LIN {X 0,Y 100.527,Z 408.465,A -85,B 0,C 180,E1 -25391.818,E2 -25391.818} C_VEL
LIN {X 0,Y 102.586,Z 414.77,A -85,B 0,C 180,E1 -25385.896,E2 -25385.896} C_VEL
LIN {X 0,Y 105.943,Z 419.989,A -85,B 0,C 180,E1 -25379.998,E2 -25379.998} C_VEL
LIN {X 0,Y 110.426,Z 424.014,A -85,B 0,C 180,E1 -25374.52,E2 -25374.52} C_VEL
LIN {X 0,Y 116.041,Z 426.901,A -85,B 0,C 180,E1 -25369.53,E2 -25369.53} C_VEL
LIN {X 0,Y 120.304,Z 428.232,A -85,B 0,C 180,E1 -25366.485,E2 -25366.485} C_VEL
LIN {X 0,Y 124.925,Z 429.078,A -85,B 0,C 180,E1 -25363.661,E2 -25363.661} C_VEL
LIN {X 0,Y 131.477,Z 429.442,A -85,B 0,C 180,E1 -25360.34,E2 -25360.34} C_VEL
LIN {X 0,Y 140.786,Z 428.809,A -85,B 0,C 180,E1 -25356.461,E2 -25356.461} C_VEL
LIN {X 0,Y 148.981,Z 427.173,A -85,B 0,C 180,E1 -25353.679,E2 -25353.679} C_VEL
LIN {X 0,Y 158.987,Z 424.026,A -85,B 0,C 180,E1 -25350.904,E2 -25350.904} C_VEL
LIN {X 0,Y 169.115,Z 419.541,A -85,B 0,C 180,E1 -25348.564,E2 -25348.564} C_VEL
LIN {X 0,Y 167.944,Z 420.358,A -85,B 0,C 180,E1 -25347.788,E2 -25347.788} C_VEL
LIN {X 0,Y 157.475,Z 425.979,A -85,B 0,C 180,E1 -25345.656,E2 -25345.656} C_VEL
LIN {X 0,Y 148.742,Z 429.762,A -85,B 0,C 180,E1 -25343.443,E2 -25343.443} C_VEL
LIN {X 0,Y 139.769,Z 432.826,A -85,B 0,C 180,E1 -25340.691,E2 -25340.691} C_VEL
LIN {X 0,Y 134.979,Z 434.073,A -85,B 0,C 180,E1 -25339.334,E2 -25339.334} C_VEL
LIN {X 0,Y 126.203,Z 435.352,A -85,B 0,C 180,E1 -25337.386,E2 -25337.386} C_VEL
LIN {X 0,Y 117.725,Z 435.788,A -85,B 0,C 180,E1 -25335.033,E2 -25335.033} C_VEL
LIN {X 0,Y 113.512,Z 435.775,A -85,B 0,C 180,E1 -25333.009,E2 -25333.009} C_VEL
LIN {X 0,Y 105.631,Z 435.098,A -85,B 0,C 180,E1 -25326.787,E2 -25326.787} C_VEL
LIN {X 0,Y 99.678,Z 433.169,A -85,B 0,C 180,E1 -25319.577,E2 -25319.577} C_VEL
LIN {X 0,Y 96.026,Z 429.965,A -85,B 0,C 180,E1 -25311.469,E2 -25311.469} C_VEL
LIN {X 0,Y 94.866,Z 425.439,A -85,B 0,C 180,E1 -25302.844,E2 -25302.844} C_VEL
LIN {X 0,Y 95.674,Z 420.934,A -85,B 0,C 180,E1 -25296.329,E2 -25296.329} C_VEL
LIN {X 0,Y 96.226,Z 419.177,A -85,B 0,C 180,E1 -25294.191,E2 -25294.191} C_VEL
LIN {X 0,Y 95.972,Z 415.73,A -85,B 0,C 180,E1 -25291.052,E2 -25291.052} C_VEL
LIN {X 0,Y 95.262,Z 408.535,A -85,B 0,C 180,E1 -25285.772,E2 -25285.772} C_VEL
LIN {X 0,Y 95.129,Z 399.527,A -85,B 0,C 180,E1 -25280.435,E2 -25280.435} C_VEL
LIN {X 0,Y 95.647,Z 389.719,A -85,B 0,C 180,E1 -25275.746,E2 -25275.746} C_VEL
LIN {X 0,Y 96.578,Z 378.914,A -85,B 0,C 180,E1 -25271.723,E2 -25271.723} C_VEL
LIN {X 0,Y 97.631,Z 367.123,A -85,B 0,C 180,E1 -25268.354,E2 -25268.354} C_VEL
LIN {X 0,Y 98.64,Z 354.886,A -85,B 0,C 180,E1 -25265.819,E2 -25265.819} C_VEL
LIN {X 0,Y 99.244,Z 342.152,A -85,B 0,C 180,E1 -25264.016,E2 -25264.016} C_VEL
LIN {X 0,Y 100.899,Z 303.926,A -85,B 0,C 180,E1 -25259.798,E2 -25259.798} C_VEL
LIN {X 0,Y 99.621,Z 267.157,A -85,B 0,C 180,E1 -25255.645,E2 -25255.645} C_VEL
LIN {X 0,Y 99.558,Z 258.226,A -85,B 0,C 180,E1 -25254.646,E2 -25254.646} C_VEL
LIN {X 0,Y 97.627,Z 250.234,A -85,B 0,C 180,E1 -25253.451,E2 -25253.451} C_VEL
LIN {X 0,Y 95.667,Z 241.869,A -85,B 0,C 180,E1 -25247.279,E2 -25247.279} C_VEL
LIN {X 0,Y 93.662,Z 232.93,A -85,B 0,C 180,E1 -25239.981,E2 -25239.981} C_VEL
LIN {X 0,Y 93.575,Z 232.827,A -85,B 0,C 180,E1 -25231.72,E2 -25231.72} C_VEL
LIN {X 0,Y 93.665,Z 232.813,A -85,B 0,C 180,E1 -25225.797,E2 -25225.797} C_VEL
LIN {X 0,Y 93.69,Z 232.814,A -85,B 0,C 180,E1 -25222.031,E2 -25222.031} C_VEL
LIN {X 0,Y 94.087,Z 232.763,A -85,B 0,C 180,E1 -25212.951,E2 -25212.951} C_VEL
LIN {X 0,Y 94.195,Z 232.749,A -85,B 0,C 180,E1 -25208.584,E2 -25208.584} C_VEL
LIN {X 0,Y 94.786,Z 232.675,A -85,B 0,C 180,E1 -25200.002,E2 -25200.002} C_VEL
LIN {X 0,Y 94.17,Z 232.753,A -85,B 0,C 180,E1 -25191.418,E2 -25191.418} C_VEL
LIN {X 0,Y 94.018,Z 232.768,A -85,B 0,C 180,E1 -25186.339,E2 -25186.339} C_VEL
LIN {X 0,Y 93.685,Z 232.809,A -85,B 0,C 180,E1 -25177.973,E2 -25177.973} C_VEL
LIN {X 0,Y 93.617,Z 232.823,A -85,B 0,C 180,E1 -25173.231,E2 -25173.231} C_VEL
LIN {X 0,Y 93.607,Z 232.825,A -85,B 0,C 180,E1 -25165.672,E2 -25165.672} C_VEL
LIN {X 0,Y 93.625,Z 232.821,A -85,B 0,C 180,E1 -25157.503,E2 -25157.503} C_VEL
LIN {X 0,Y 93.623,Z 232.815,A -85,B 0,C 180,E1 -25151.355,E2 -25151.355} C_VEL
LIN {X 0,Y 93.609,Z 232.818,A -85,B 0,C 180,E1 -25144.328,E2 -25144.328} C_VEL
LIN {X 0,Y 93.665,Z 232.812,A -85,B 0,C 180,E1 -25135.794,E2 -25135.794} C_VEL
LIN {X 0,Y 93.689,Z 232.814,A -85,B 0,C 180,E1 -25132.025,E2 -25132.025} C_VEL
LIN {X 0,Y 94.088,Z 232.765,A -85,B 0,C 180,E1 -25122.946,E2 -25122.946} C_VEL
LIN {X 0,Y 94.197,Z 232.744,A -85,B 0,C 180,E1 -25118.579,E2 -25118.579} C_VEL
LIN {X 0,Y 94.794,Z 232.67,A -85,B 0,C 180,E1 -25109.997,E2 -25109.997} C_VEL
LIN {X 0,Y 94.209,Z 232.743,A -85,B 0,C 180,E1 -25101.416,E2 -25101.416} C_VEL
LIN {X 0,Y 94.045,Z 232.77,A -85,B 0,C 180,E1 -25096.276,E2 -25096.276} C_VEL
LIN {X 0,Y 93.692,Z 232.812,A -85,B 0,C 180,E1 -25087.969,E2 -25087.969} C_VEL
LIN {X 0,Y 93.813,Z 232.951,A -85,B 0,C 180,E1 -25080.549,E2 -25080.549} C_VEL
LIN {X 0,Y 94.861,Z 237.645,A -85,B 0,C 180,E1 -25076.331,E2 -25076.331} C_VEL
LIN {X 0,Y 95.705,Z 241.642,A -85,B 0,C 180,E1 -25073.185,E2 -25073.185} C_VEL
LIN {X 0,Y 100.113,Z 259.74,A -85,B 0,C 180,E1 -25070.488,E2 -25070.488} C_VEL
LIN {X 0,Y 101.197,Z 271.435,A -85,B 0,C 180,E1 -25069.044,E2 -25069.044} C_VEL
LIN {X 0,Y 97.514,Z 333.744,A -85,B 0,C 180,E1 -25061.785,E2 -25061.785} C_VEL
LIN {X 0,Y 96.446,Z 347.717,A -85,B 0,C 180,E1 -25059.273,E2 -25059.273} C_VEL
LIN {X 0,Y 95.268,Z 359.841,A -85,B 0,C 180,E1 -25056.166,E2 -25056.166} C_VEL
LIN {X 0,Y 94.062,Z 371.748,A -85,B 0,C 180,E1 -25052.089,E2 -25052.089} C_VEL
LIN {X 0,Y 93.221,Z 382.27,A -85,B 0,C 180,E1 -25047.499,E2 -25047.499} C_VEL
LIN {X 0,Y 92.756,Z 391.836,A -85,B 0,C 180,E1 -25042.26,E2 -25042.26} C_VEL
LIN {X 0,Y 92.8,Z 400.424,A -85,B 0,C 180,E1 -25036.497,E2 -25036.497} C_VEL
LIN {X 0,Y 93.861,Z 407.958,A -85,B 0,C 180,E1 -25030.304,E2 -25030.304} C_VEL
LIN {X 0,Y 96.102,Z 414.282,A -85,B 0,C 180,E1 -25024.192,E2 -25024.192} C_VEL
LIN {X 0,Y 99.787,Z 419.82,A -85,B 0,C 180,E1 -25017.98,E2 -25017.98} C_VEL
LIN {X 0,Y 104.629,Z 424.049,A -85,B 0,C 180,E1 -25012.278,E2 -25012.278} C_VEL
LIN {X 0,Y 108.524,Z 426.246,A -85,B 0,C 180,E1 -25008.796,E2 -25008.796} C_VEL
LIN {X 0,Y 112.895,Z 428.007,A -85,B 0,C 180,E1 -25005.579,E2 -25005.579} C_VEL
LIN {X 0,Y 117.979,Z 429.323,A -85,B 0,C 180,E1 -25002.392,E2 -25002.392} C_VEL
LIN {X 0,Y 126.464,Z 430.273,A -85,B 0,C 180,E1 -24998.15,E2 -24998.15} C_VEL
LIN {X 0,Y 133.801,Z 430.216,A -85,B 0,C 180,E1 -24995.151,E2 -24995.151} C_VEL
LIN {X 0,Y 143.305,Z 429.03,A -85,B 0,C 180,E1 -24991.98,E2 -24991.98} C_VEL
LIN {X 0,Y 152.344,Z 426.875,A -85,B 0,C 180,E1 -24989.504,E2 -24989.504} C_VEL
LIN {X 0,Y 156.663,Z 425.494,A -85,B 0,C 180,E1 -24988.471,E2 -24988.471} C_VEL
LIN {X 0,Y 144.639,Z 430.196,A -85,B 0,C 180,E1 -24985.696,E2 -24985.696} C_VEL
LIN {X 0,Y 133.24,Z 433.412,A -85,B 0,C 180,E1 -24982.301,E2 -24982.301} C_VEL
LIN {X 0,Y 122.723,Z 435.225,A -85,B 0,C 180,E1 -24978.117,E2 -24978.117} C_VEL
LIN {X 0,Y 113.512,Z 435.775,A -85,B 0,C 180,E1 -24973.009,E2 -24973.009} C_VEL
LIN {X 0,Y 109.506,Z 435.577,A -85,B 0,C 180,E1 -24970.776,E2 -24970.776} C_VEL
LIN {X 0,Y 102.13,Z 434.213,A -85,B 0,C 180,E1 -24967.256,E2 -24967.256} C_VEL
LIN {X 0,Y 95.497,Z 432.125,A -85,B 0,C 180,E1 -24963.169,E2 -24963.169} C_VEL
LIN {X 0,Y 92.799,Z 430.741,A -85,B 0,C 180,E1 -24960.084,E2 -24960.084} C_VEL
LIN {X 0,Y 89.119,Z 426.724,A -85,B 0,C 180,E1 -24950.789,E2 -24950.789} C_VEL
LIN {X 0,Y 88.499,Z 421.402,A -85,B 0,C 180,E1 -24941.454,E2 -24941.454} C_VEL
LIN {X 0,Y 89.676,Z 416.276,A -85,B 0,C 180,E1 -24934.498,E2 -24934.498} C_VEL
LIN {X 0,Y 89.047,Z 411.079,A -85,B 0,C 180,E1 -24930.003,E2 -24930.003} C_VEL
LIN {X 0,Y 88.409,Z 402.899,A -85,B 0,C 180,E1 -24924.301,E2 -24924.301} C_VEL
LIN {X 0,Y 88.508,Z 392.727,A -85,B 0,C 180,E1 -24918.553,E2 -24918.553} C_VEL
LIN {X 0,Y 89.198,Z 382.49,A -85,B 0,C 180,E1 -24913.996,E2 -24913.996} C_VEL
LIN {X 0,Y 90.216,Z 370.996,A -85,B 0,C 180,E1 -24910.003,E2 -24910.003} C_VEL
LIN {X 0,Y 91.441,Z 357.072,A -85,B 0,C 180,E1 -24906.507,E2 -24906.507} C_VEL
LIN {X 0,Y 92.057,Z 344.663,A -85,B 0,C 180,E1 -24904.421,E2 -24904.421} C_VEL
LIN {X 0,Y 93.823,Z 304.102,A -85,B 0,C 180,E1 -24899.536,E2 -24899.536} C_VEL
LIN {X 0,Y 92.573,Z 267.775,A -85,B 0,C 180,E1 -24895.12,E2 -24895.12} C_VEL
LIN {X 0,Y 92.653,Z 259.76,A -85,B 0,C 180,E1 -24894.166,E2 -24894.166} C_VEL
LIN {X 0,Y 90.29,Z 249.862,A -85,B 0,C 180,E1 -24892.583,E2 -24892.583} C_VEL
LIN {X 0,Y 88.272,Z 241.356,A -85,B 0,C 180,E1 -24885.774,E2 -24885.774} C_VEL
LIN {X 0,Y 86.553,Z 233.814,A -85,B 0,C 180,E1 -24878.989,E2 -24878.989} C_VEL
LIN {X 0,Y 86.53,Z 233.708,A -85,B 0,C 180,E1 -24874.651,E2 -24874.651} C_VEL
LIN {X 0,Y 86.579,Z 233.693,A -85,B 0,C 180,E1 -24866.767,E2 -24866.767} C_VEL
LIN {X 0,Y 86.643,Z 233.684,A -85,B 0,C 180,E1 -24858.935,E2 -24858.935} C_VEL
LIN {X 0,Y 86.965,Z 233.652,A -85,B 0,C 180,E1 -24854.033,E2 -24854.033} C_VEL
LIN {X 0,Y 87.103,Z 233.629,A -85,B 0,C 180,E1 -24849.289,E2 -24849.289} C_VEL
LIN {X 0,Y 87.713,Z 233.556,A -85,B 0,C 180,E1 -24840.002,E2 -24840.002} C_VEL
LIN {X 0,Y 87.08,Z 233.637,A -85,B 0,C 180,E1 -24830.713,E2 -24830.713} C_VEL
LIN {X 0,Y 86.925,Z 233.65,A -85,B 0,C 180,E1 -24825.965,E2 -24825.965} C_VEL
LIN {X 0,Y 86.638,Z 233.693,A -85,B 0,C 180,E1 -24821.069,E2 -24821.069} C_VEL
LIN {X 0,Y 86.579,Z 233.7,A -85,B 0,C 180,E1 -24813.233,E2 -24813.233} C_VEL
LIN {X 0,Y 86.531,Z 233.707,A -85,B 0,C 180,E1 -24804.305,E2 -24804.305} C_VEL
LIN {X 0,Y 86.553,Z 233.703,A -85,B 0,C 180,E1 -24796.947,E2 -24796.947} C_VEL
LIN {X 0,Y 86.548,Z 233.698,A -85,B 0,C 180,E1 -24790.509,E2 -24790.509} C_VEL
LIN {X 0,Y 86.556,Z 233.697,A -85,B 0,C 180,E1 -24784.632,E2 -24784.632} C_VEL
LIN {X 0,Y 86.581,Z 233.696,A -85,B 0,C 180,E1 -24776.765,E2 -24776.765} C_VEL
LIN {X 0,Y 86.658,Z 233.688,A -85,B 0,C 180,E1 -24768.926,E2 -24768.926} C_VEL
LIN {X 0,Y 86.966,Z 233.651,A -85,B 0,C 180,E1 -24764.027,E2 -24764.027} C_VEL
LIN {X 0,Y 87.105,Z 233.629,A -85,B 0,C 180,E1 -24759.283,E2 -24759.283} C_VEL
LIN {X 0,Y 87.721,Z 233.55,A -85,B 0,C 180,E1 -24749.997,E2 -24749.997} C_VEL
LIN {X 0,Y 87.115,Z 233.626,A -85,B 0,C 180,E1 -24740.712,E2 -24740.712} C_VEL
LIN {X 0,Y 86.949,Z 233.654,A -85,B 0,C 180,E1 -24735.909,E2 -24735.909} C_VEL
LIN {X 0,Y 86.662,Z 233.69,A -85,B 0,C 180,E1 -24731.068,E2 -24731.068} C_VEL
LIN {X 0,Y 86.708,Z 233.721,A -85,B 0,C 180,E1 -24721.757,E2 -24721.757} C_VEL
LIN {X 0,Y 86.974,Z 234.779,A -85,B 0,C 180,E1 -24720.331,E2 -24720.331} C_VEL
LIN {X 0,Y 88.541,Z 241.92,A -85,B 0,C 180,E1 -24714.05,E2 -24714.05} C_VEL
LIN {X 0,Y 93.165,Z 260.956,A -85,B 0,C 180,E1 -24710.987,E2 -24710.987} C_VEL
LIN {X 0,Y 94.057,Z 272.878,A -85,B 0,C 180,E1 -24709.439,E2 -24709.439} C_VEL
LIN {X 0,Y 90.386,Z 334.333,A -85,B 0,C 180,E1 -24701.646,E2 -24701.646} C_VEL
LIN {X 0,Y 89.315,Z 347.777,A -85,B 0,C 180,E1 -24699.011,E2 -24699.011} C_VEL
LIN {X 0,Y 88.063,Z 360.548,A -85,B 0,C 180,E1 -24695.448,E2 -24695.448} C_VEL
LIN {X 0,Y 86.936,Z 372.452,A -85,B 0,C 180,E1 -24691.019,E2 -24691.019} C_VEL
LIN {X 0,Y 86.193,Z 382.575,A -85,B 0,C 180,E1 -24686.238,E2 -24686.238} C_VEL
LIN {X 0,Y 85.855,Z 390.572,A -85,B 0,C 180,E1 -24681.612,E2 -24681.612} C_VEL
LIN {X 0,Y 86.125,Z 400.857,A -85,B 0,C 180,E1 -24674.168,E2 -24674.168} C_VEL
LIN {X 0,Y 87.827,Z 409.128,A -85,B 0,C 180,E1 -24666.892,E2 -24666.892} C_VEL
LIN {X 0,Y 90.949,Z 415.817,A -85,B 0,C 180,E1 -24659.998,E2 -24659.998} C_VEL
LIN {X 0,Y 95.39,Z 421.11,A -85,B 0,C 180,E1 -24653.653,E2 -24653.653} C_VEL
LIN {X 0,Y 101.091,Z 425.24,A -85,B 0,C 180,E1 -24647.96,E2 -24647.96} C_VEL
LIN {X 0,Y 105.481,Z 427.38,A -85,B 0,C 180,E1 -24644.541,E2 -24644.541} C_VEL
LIN {X 0,Y 111.809,Z 429.446,A -85,B 0,C 180,E1 -24640.543,E2 -24640.543} C_VEL
LIN {X 0,Y 121.658,Z 431.046,A -85,B 0,C 180,E1 -24635.765,E2 -24635.765} C_VEL
LIN {X 0,Y 126.882,Z 431.269,A -85,B 0,C 180,E1 -24633.695,E2 -24633.695} C_VEL
LIN {X 0,Y 137.831,Z 430.624,A -85,B 0,C 180,E1 -24630.095,E2 -24630.095} C_VEL
LIN {X 0,Y 142.117,Z 429.979,A -85,B 0,C 180,E1 -24628.902,E2 -24628.902} C_VEL
LIN {X 0,Y 140.774,Z 430.471,A -85,B 0,C 180,E1 -24628.074,E2 -24628.074} C_VEL
LIN {X 0,Y 129.039,Z 433.206,A -85,B 0,C 180,E1 -24624.785,E2 -24624.785} C_VEL
LIN {X 0,Y 118.12,Z 434.581,A -85,B 0,C 180,E1 -24620.671,E2 -24620.671} C_VEL
LIN {X 0,Y 108.003,Z 434.667,A -85,B 0,C 180,E1 -24615.247,E2 -24615.247} C_VEL
LIN {X 0,Y 100.128,Z 433.644,A -85,B 0,C 180,E1 -24609.179,E2 -24609.179} C_VEL
LIN {X 0,Y 93.747,Z 431.355,A -85,B 0,C 180,E1 -24601.656,E2 -24601.656} C_VEL
LIN {X 0,Y 92.799,Z 430.741,A -85,B 0,C 180,E1 -24600.084,E2 -24600.084} C_VEL
LIN {X 0,Y 90.51,Z 429.227,A -85,B 0,C 180,E1 -24596.832,E2 -24596.832} C_VEL
LIN {X 0,Y 86.053,Z 425.576,A -85,B 0,C 180,E1 -24591.595,E2 -24591.595} C_VEL
LIN {X 0,Y 82.643,Z 421.188,A -85,B 0,C 180,E1 -24585.977,E2 -24585.977} C_VEL
LIN {X 0,Y 82.108,Z 418.58,A -85,B 0,C 180,E1 -24582.287,E2 -24582.287} C_VEL
LIN {X 0,Y 83.036,Z 414.21,A -85,B 0,C 180,E1 -24576.076,E2 -24576.076} C_VEL
LIN {X 0,Y 83.145,Z 413.131,A -85,B 0,C 180,E1 -24574.852,E2 -24574.852} C_VEL
LIN {X 0,Y 82.097,Z 405.873,A -85,B 0,C 180,E1 -24568.777,E2 -24568.777} C_VEL
LIN {X 0,Y 81.633,Z 396.676,A -85,B 0,C 180,E1 -24562.584,E2 -24562.584} C_VEL
LIN {X 0,Y 81.996,Z 386.295,A -85,B 0,C 180,E1 -24557.001,E2 -24557.001} C_VEL
LIN {X 0,Y 82.86,Z 374.567,A -85,B 0,C 180,E1 -24552.097,E2 -24552.097} C_VEL
LIN {X 0,Y 83.967,Z 361.337,A -85,B 0,C 180,E1 -24548.031,E2 -24548.031} C_VEL
LIN {X 0,Y 84.765,Z 349.696,A -85,B 0,C 180,E1 -24545.512,E2 -24545.512} C_VEL
LIN {X 0,Y 86.102,Z 319.784,A -85,B 0,C 180,E1 -24541.349,E2 -24541.349} C_VEL
LIN {X 0,Y 86.708,Z 303.454,A -85,B 0,C 180,E1 -24539.23,E2 -24539.23} C_VEL
LIN {X 0,Y 85.561,Z 268.314,A -85,B 0,C 180,E1 -24534.582,E2 -24534.582} C_VEL
LIN {X 0,Y 85.542,Z 260.373,A -85,B 0,C 180,E1 -24533.547,E2 -24533.547} C_VEL
LIN {X 0,Y 82.924,Z 249.539,A -85,B 0,C 180,E1 -24531.665,E2 -24531.665} C_VEL
LIN {X 0,Y 80.902,Z 240.896,A -85,B 0,C 180,E1 -24524.028,E2 -24524.028} C_VEL
LIN {X 0,Y 79.486,Z 234.684,A -85,B 0,C 180,E1 -24517.876,E2 -24517.876} C_VEL
LIN {X 0,Y 79.477,Z 234.578,A -85,B 0,C 180,E1 -24507.845,E2 -24507.845} C_VEL
LIN {X 0,Y 79.51,Z 234.577,A -85,B 0,C 180,E1 -24500.708,E2 -24500.708} C_VEL
LIN {X 0,Y 79.837,Z 234.54,A -85,B 0,C 180,E1 -24494.477,E2 -24494.477} C_VEL
LIN {X 0,Y 79.989,Z 234.513,A -85,B 0,C 180,E1 -24490.123,E2 -24490.123} C_VEL
LIN {X 0,Y 80.64,Z 234.437,A -85,B 0,C 180,E1 -24480.002,E2 -24480.002} C_VEL
LIN {X 0,Y 79.962,Z 234.525,A -85,B 0,C 180,E1 -24469.878,E2 -24469.878} C_VEL
LIN {X 0,Y 79.738,Z 234.545,A -85,B 0,C 180,E1 -24464.67,E2 -24464.67} C_VEL
LIN {X 0,Y 79.506,Z 234.579,A -85,B 0,C 180,E1 -24459.296,E2 -24459.296} C_VEL
LIN {X 0,Y 79.478,Z 234.585,A -85,B 0,C 180,E1 -24452.153,E2 -24452.153} C_VEL
LIN {X 0,Y 79.441,Z 234.588,A -85,B 0,C 180,E1 -24442.763,E2 -24442.763} C_VEL
LIN {X 0,Y 79.461,Z 234.587,A -85,B 0,C 180,E1 -24434.966,E2 -24434.966} C_VEL
LIN {X 0,Y 79.447,Z 234.589,A -85,B 0,C 180,E1 -24427.24,E2 -24427.24} C_VEL
LIN {X 0,Y 79.48,Z 234.584,A -85,B 0,C 180,E1 -24417.846,E2 -24417.846} C_VEL
LIN {X 0,Y 79.518,Z 234.581,A -85,B 0,C 180,E1 -24410.699,E2 -24410.699} C_VEL
LIN {X 0,Y 79.838,Z 234.536,A -85,B 0,C 180,E1 -24404.472,E2 -24404.472} C_VEL
LIN {X 0,Y 79.99,Z 234.518,A -85,B 0,C 180,E1 -24400.117,E2 -24400.117} C_VEL
LIN {X 0,Y 80.649,Z 234.431,A -85,B 0,C 180,E1 -24389.996,E2 -24389.996} C_VEL
LIN {X 0,Y 79.998,Z 234.515,A -85,B 0,C 180,E1 -24379.877,E2 -24379.877} C_VEL
LIN {X 0,Y 79.764,Z 234.546,A -85,B 0,C 180,E1 -24374.669,E2 -24374.669} C_VEL
LIN {X 0,Y 79.527,Z 234.579,A -85,B 0,C 180,E1 -24369.296,E2 -24369.296} C_VEL
LIN {X 0,Y 79.677,Z 234.756,A -85,B 0,C 180,E1 -24362.426,E2 -24362.426} C_VEL
LIN {X 0,Y 81.142,Z 241.312,A -85,B 0,C 180,E1 -24355.733,E2 -24355.733} C_VEL
LIN {X 0,Y 81.37,Z 242.366,A -85,B 0,C 180,E1 -24354.903,E2 -24354.903} C_VEL
LIN {X 0,Y 86.246,Z 262.636,A -85,B 0,C 180,E1 -24351.415,E2 -24351.415} C_VEL
LIN {X 0,Y 87.016,Z 272.556,A -85,B 0,C 180,E1 -24350.008,E2 -24350.008} C_VEL
LIN {X 0,Y 83.263,Z 335.069,A -85,B 0,C 180,E1 -24341.377,E2 -24341.377} C_VEL
LIN {X 0,Y 82.113,Z 348.391,A -85,B 0,C 180,E1 -24338.523,E2 -24338.523} C_VEL
LIN {X 0,Y 81.013,Z 359.879,A -85,B 0,C 180,E1 -24335.078,E2 -24335.078} C_VEL
LIN {X 0,Y 79.964,Z 371.507,A -85,B 0,C 180,E1 -24330.519,E2 -24330.519} C_VEL
LIN {X 0,Y 79.257,Z 382.434,A -85,B 0,C 180,E1 -24324.907,E2 -24324.907} C_VEL
LIN {X 0,Y 78.947,Z 390.93,A -85,B 0,C 180,E1 -24319.499,E2 -24319.499} C_VEL
LIN {X 0,Y 79.536,Z 400.525,A -85,B 0,C 180,E1 -24312.087,E2 -24312.087} C_VEL
LIN {X 0,Y 81.361,Z 408.296,A -85,B 0,C 180,E1 -24304.953,E2 -24304.953} C_VEL
LIN {X 0,Y 85.331,Z 415.854,A -85,B 0,C 180,E1 -24296.872,E2 -24296.872} C_VEL
LIN {X 0,Y 89.703,Z 420.771,A -85,B 0,C 180,E1 -24290.983,E2 -24290.983} C_VEL
LIN {X 0,Y 95.944,Z 425.213,A -85,B 0,C 180,E1 -24285.057,E2 -24285.057} C_VEL
LIN {X 0,Y 103.095,Z 428.47,A -85,B 0,C 180,E1 -24280.069,E2 -24280.069} C_VEL
LIN {X 0,Y 108.366,Z 430.078,A -85,B 0,C 180,E1 -24277.098,E2 -24277.098} C_VEL
LIN {X 0,Y 118.859,Z 431.845,A -85,B 0,C 180,E1 -24272.494,E2 -24272.494} C_VEL
LIN {X 0,Y 128.984,Z 432.154,A -85,B 0,C 180,E1 -24269.065,E2 -24269.065} C_VEL
LIN {X 0,Y 128.114,Z 432.417,A -85,B 0,C 180,E1 -24268.305,E2 -24268.305} C_VEL
LIN {X 0,Y 119.296,Z 433.468,A -85,B 0,C 180,E1 -24265.569,E2 -24265.569} C_VEL
LIN {X 0,Y 108.537,Z 433.792,A -85,B 0,C 180,E1 -24260.992,E2 -24260.992} C_VEL
LIN {X 0,Y 99.039,Z 432.908,A -85,B 0,C 180,E1 -24255.207,E2 -24255.207} C_VEL
LIN {X 0,Y 91.16,Z 430.864,A -85,B 0,C 180,E1 -24248.084,E2 -24248.084} C_VEL
LIN {X 0,Y 85.449,Z 427.598,A -85,B 0,C 180,E1 -24239.573,E2 -24239.573} C_VEL
LIN {X 0,Y 82.404,Z 423.04,A -85,B 0,C 180,E1 -24229.95,E2 -24229.95} C_VEL
LIN {X 0,Y 82.108,Z 418.58,A -85,B 0,C 180,E1 -24222.287,E2 -24222.287} C_VEL
LIN {X 0,Y 81.96,Z 416.788,A -85,B 0,C 180,E1 -24219.899,E2 -24219.899} C_VEL
LIN {X 0,Y 81.28,Z 414.6,A -85,B 0,C 180,E1 -24217.675,E2 -24217.675} C_VEL
LIN {X 0,Y 79.644,Z 410.864,A -85,B 0,C 180,E1 -24214.59,E2 -24214.59} C_VEL
LIN {X 0,Y 75.525,Z 400.581,A -85,B 0,C 180,E1 -24207.668,E2 -24207.668} C_VEL
LIN {X 0,Y 75.066,Z 397.473,A -85,B 0,C 180,E1 -24205.585,E2 -24205.585} C_VEL
LIN {X 0,Y 75.076,Z 387.142,A -85,B 0,C 180,E1 -24199.213,E2 -24199.213} C_VEL
LIN {X 0,Y 75.735,Z 375.961,A -85,B 0,C 180,E1 -24193.84,E2 -24193.84} C_VEL
LIN {X 0,Y 76.669,Z 364.055,A -85,B 0,C 180,E1 -24189.549,E2 -24189.549} C_VEL
LIN {X 0,Y 77.501,Z 352.51,A -85,B 0,C 180,E1 -24186.516,E2 -24186.516} C_VEL
LIN {X 0,Y 78.112,Z 339.079,A -85,B 0,C 180,E1 -24184.129,E2 -24184.129} C_VEL
LIN {X 0,Y 79.659,Z 304.435,A -85,B 0,C 180,E1 -24179.153,E2 -24179.153} C_VEL
LIN {X 0,Y 78.522,Z 268.388,A -85,B 0,C 180,E1 -24173.937,E2 -24173.937} C_VEL
LIN {X 0,Y 78.489,Z 261.196,A -85,B 0,C 180,E1 -24172.893,E2 -24172.893} C_VEL
LIN {X 0,Y 75.592,Z 249.161,A -85,B 0,C 180,E1 -24170.609,E2 -24170.609} C_VEL
LIN {X 0,Y 73.516,Z 240.36,A -85,B 0,C 180,E1 -24162.008,E2 -24162.008} C_VEL
LIN {X 0,Y 72.385,Z 235.556,A -85,B 0,C 180,E1 -24156.624,E2 -24156.624} C_VEL
LIN {X 0,Y 72.372,Z 235.467,A -85,B 0,C 180,E1 -24149.051,E2 -24149.051} C_VEL
LIN {X 0,Y 72.39,Z 235.468,A -85,B 0,C 180,E1 -24142.854,E2 -24142.854} C_VEL
LIN {X 0,Y 72.732,Z 235.425,A -85,B 0,C 180,E1 -24134.937,E2 -24134.937} C_VEL
LIN {X 0,Y 72.875,Z 235.399,A -85,B 0,C 180,E1 -24131.123,E2 -24131.123} C_VEL
LIN {X 0,Y 73.566,Z 235.318,A -85,B 0,C 180,E1 -24120.003,E2 -24120.003} C_VEL
LIN {X 0,Y 72.853,Z 235.41,A -85,B 0,C 180,E1 -24108.879,E2 -24108.879} C_VEL
LIN {X 0,Y 72.567,Z 235.443,A -85,B 0,C 180,E1 -24103.112,E2 -24103.112} C_VEL
LIN {X 0,Y 72.387,Z 235.459,A -85,B 0,C 180,E1 -24097.151,E2 -24097.151} C_VEL
LIN {X 0,Y 72.37,Z 235.468,A -85,B 0,C 180,E1 -24090.918,E2 -24090.918} C_VEL
LIN {X 0,Y 72.329,Z 235.476,A -85,B 0,C 180,E1 -24084.341,E2 -24084.341} C_VEL
LIN {X 0,Y 72.304,Z 235.477,A -85,B 0,C 180,E1 -24077.129,E2 -24077.129} C_VEL
LIN {X 0,Y 72.354,Z 235.471,A -85,B 0,C 180,E1 -24069.011,E2 -24069.011} C_VEL
LIN {X 0,Y 72.333,Z 235.473,A -85,B 0,C 180,E1 -24065.654,E2 -24065.654} C_VEL
LIN {X 0,Y 72.387,Z 235.468,A -85,B 0,C 180,E1 -24059.037,E2 -24059.037} C_VEL
LIN {X 0,Y 72.395,Z 235.463,A -85,B 0,C 180,E1 -24052.845,E2 -24052.845} C_VEL
LIN {X 0,Y 72.753,Z 235.417,A -85,B 0,C 180,E1 -24044.993,E2 -24044.993} C_VEL
LIN {X 0,Y 72.876,Z 235.406,A -85,B 0,C 180,E1 -24041.116,E2 -24041.116} C_VEL
LIN {X 0,Y 73.575,Z 235.312,A -85,B 0,C 180,E1 -24029.996,E2 -24029.996} C_VEL
LIN {X 0,Y 72.883,Z 235.404,A -85,B 0,C 180,E1 -24018.877,E2 -24018.877} C_VEL
LIN {X 0,Y 72.586,Z 235.437,A -85,B 0,C 180,E1 -24013.11,E2 -24013.11} C_VEL
LIN {X 0,Y 72.567,Z 235.569,A -85,B 0,C 180,E1 -24003.773,E2 -24003.773} C_VEL
LIN {X 0,Y 73.029,Z 237.535,A -85,B 0,C 180,E1 -24001.234,E2 -24001.234} C_VEL
LIN {X 0,Y 74.194,Z 242.699,A -85,B 0,C 180,E1 -23995.933,E2 -23995.933} C_VEL
LIN {X 0,Y 79.335,Z 264.278,A -85,B 0,C 180,E1 -23991.874,E2 -23991.874} C_VEL
LIN {X 0,Y 79.893,Z 273.059,A -85,B 0,C 180,E1 -23990.524,E2 -23990.524} C_VEL
LIN {X 0,Y 76.195,Z 334.708,A -85,B 0,C 180,E1 -23981.263,E2 -23981.263} C_VEL
LIN {X 0,Y 75.091,Z 347.518,A -85,B 0,C 180,E1 -23978.317,E2 -23978.317} C_VEL
LIN {X 0,Y 73.926,Z 359.791,A -85,B 0,C 180,E1 -23974.321,E2 -23974.321} C_VEL
LIN {X 0,Y 72.883,Z 372.355,A -85,B 0,C 180,E1 -23968.822,E2 -23968.822} C_VEL
LIN {X 0,Y 72.315,Z 384.067,A -85,B 0,C 180,E1 -23962.12,E2 -23962.12} C_VEL
LIN {X 0,Y 72.451,Z 395.051,A -85,B 0,C 180,E1 -23954.047,E2 -23954.047} C_VEL
LIN {X 0,Y 74.106,Z 404.498,A -85,B 0,C 180,E1 -23945.439,E2 -23945.439} C_VEL
LIN {X 0,Y 77.82,Z 412.82,A -85,B 0,C 180,E1 -23936.764,E2 -23936.764} C_VEL
LIN {X 0,Y 82.314,Z 418.513,A -85,B 0,C 180,E1 -23930.166,E2 -23930.166} C_VEL
LIN {X 0,Y 89.104,Z 423.897,A -85,B 0,C 180,E1 -23923.399,E2 -23923.399} C_VEL
LIN {X 0,Y 95.903,Z 427.478,A -85,B 0,C 180,E1 -23918.503,E2 -23918.503} C_VEL
LIN {X 0,Y 101.339,Z 429.524,A -85,B 0,C 180,E1 -23915.409,E2 -23915.409} C_VEL
LIN {X 0,Y 107.145,Z 431.077,A -85,B 0,C 180,E1 -23912.665,E2 -23912.665} C_VEL
LIN {X 0,Y 113.45,Z 432.245,A -85,B 0,C 180,E1 -23910.147,E2 -23910.147} C_VEL
LIN {X 0,Y 115.46,Z 432.721,A -85,B 0,C 180,E1 -23908.453,E2 -23908.453} C_VEL
LIN {X 0,Y 104.276,Z 432.624,A -85,B 0,C 180,E1 -23903.98,E2 -23903.98} C_VEL
LIN {X 0,Y 94.273,Z 431.367,A -85,B 0,C 180,E1 -23898.206,E2 -23898.206} C_VEL
LIN {X 0,Y 85.882,Z 428.907,A -85,B 0,C 180,E1 -23890.898,E2 -23890.898} C_VEL
LIN {X 0,Y 79.65,Z 425.291,A -85,B 0,C 180,E1 -23881.97,E2 -23881.97} C_VEL
LIN {X 0,Y 76.23,Z 420.334,A -85,B 0,C 180,E1 -23871.644,E2 -23871.644} C_VEL
LIN {X 0,Y 75.807,Z 415.511,A -85,B 0,C 180,E1 -23863.089,E2 -23863.089} C_VEL
LIN {X 0,Y 76.716,Z 410.967,A -85,B 0,C 180,E1 -23856.579,E2 -23856.579} C_VEL
LIN {X 0,Y 75.774,Z 405.137,A -85,B 0,C 180,E1 -23851.332,E2 -23851.332} C_VEL
LIN {X 0,Y 75.066,Z 397.473,A -85,B 0,C 180,E1 -23845.585,E2 -23845.585} C_VEL
LIN {X 0,Y 74.33,Z 392.909,A -85,B 0,C 180,E1 -23842.82,E2 -23842.82} C_VEL
LIN {X 0,Y 72.905,Z 388.046,A -85,B 0,C 180,E1 -23840.423,E2 -23840.423} C_VEL
LIN {X 0,Y 69.477,Z 376.059,A -85,B 0,C 180,E1 -23835.365,E2 -23835.365} C_VEL
LIN {X 0,Y 69.165,Z 370.632,A -85,B 0,C 180,E1 -23833.148,E2 -23833.148} C_VEL
LIN {X 0,Y 70.01,Z 359.201,A -85,B 0,C 180,E1 -23829.05,E2 -23829.05} C_VEL
LIN {X 0,Y 70.722,Z 347.421,A -85,B 0,C 180,E1 -23826.028,E2 -23826.028} C_VEL
LIN {X 0,Y 72.581,Z 304.67,A -85,B 0,C 180,E1 -23818.971,E2 -23818.971} C_VEL
LIN {X 0,Y 71.485,Z 268.942,A -85,B 0,C 180,E1 -23813.324,E2 -23813.324} C_VEL
LIN {X 0,Y 71.477,Z 262.238,A -85,B 0,C 180,E1 -23812.269,E2 -23812.269} C_VEL
LIN {X 0,Y 68.247,Z 248.92,A -85,B 0,C 180,E1 -23809.475,E2 -23809.475} C_VEL
LIN {X 0,Y 66.128,Z 239.886,A -85,B 0,C 180,E1 -23799.622,E2 -23799.622} C_VEL
LIN {X 0,Y 65.267,Z 236.437,A -85,B 0,C 180,E1 -23795.132,E2 -23795.132} C_VEL
LIN {X 0,Y 65.257,Z 236.357,A -85,B 0,C 180,E1 -23790.516,E2 -23790.516} C_VEL
LIN {X 0,Y 65.234,Z 236.354,A -85,B 0,C 180,E1 -23785.53,E2 -23785.53} C_VEL
LIN {X 0,Y 65.632,Z 236.309,A -85,B 0,C 180,E1 -23775.496,E2 -23775.496} C_VEL
LIN {X 0,Y 65.768,Z 236.288,A -85,B 0,C 180,E1 -23772.343,E2 -23772.343} C_VEL
LIN {X 0,Y 66.489,Z 236.199,A -85,B 0,C 180,E1 -23760.003,E2 -23760.003} C_VEL
LIN {X 0,Y 65.749,Z 236.292,A -85,B 0,C 180,E1 -23747.659,E2 -23747.659} C_VEL
LIN {X 0,Y 65.374,Z 236.342,A -85,B 0,C 180,E1 -23741.188,E2 -23741.188} C_VEL
LIN {X 0,Y 65.24,Z 236.356,A -85,B 0,C 180,E1 -23734.479,E2 -23734.479} C_VEL
LIN {X 0,Y 65.208,Z 236.355,A -85,B 0,C 180,E1 -23727.395,E2 -23727.395} C_VEL
LIN {X 0,Y 65.238,Z 236.352,A -85,B 0,C 180,E1 -23718.939,E2 -23718.939} C_VEL
LIN {X 0,Y 65.262,Z 236.349,A -85,B 0,C 180,E1 -23710.245,E2 -23710.245} C_VEL
LIN {X 0,Y 65.255,Z 236.355,A -85,B 0,C 180,E1 -23700.509,E2 -23700.509} C_VEL
LIN {X 0,Y 65.244,Z 236.35,A -85,B 0,C 180,E1 -23695.518,E2 -23695.518} C_VEL
LIN {X 0,Y 65.647,Z 236.3,A -85,B 0,C 180,E1 -23685.536,E2 -23685.536} C_VEL
LIN {X 0,Y 65.777,Z 236.292,A -85,B 0,C 180,E1 -23682.334,E2 -23682.334} C_VEL
LIN {X 0,Y 66.499,Z 236.193,A -85,B 0,C 180,E1 -23669.996,E2 -23669.996} C_VEL
LIN {X 0,Y 65.782,Z 236.291,A -85,B 0,C 180,E1 -23657.658,E2 -23657.658} C_VEL
LIN {X 0,Y 65.4,Z 236.337,A -85,B 0,C 180,E1 -23651.188,E2 -23651.188} C_VEL
LIN {X 0,Y 65.421,Z 236.379,A -85,B 0,C 180,E1 -23645.396,E2 -23645.396} C_VEL
LIN {X 0,Y 65.822,Z 237.852,A -85,B 0,C 180,E1 -23643.009,E2 -23643.009} C_VEL
LIN {X 0,Y 67.04,Z 243.06,A -85,B 0,C 180,E1 -23637.051,E2 -23637.051} C_VEL
LIN {X 0,Y 72.333,Z 265.182,A -85,B 0,C 180,E1 -23632.473,E2 -23632.473} C_VEL
LIN {X 0,Y 72.854,Z 273.008,A -85,B 0,C 180,E1 -23631.17,E2 -23631.17} C_VEL
LIN {X 0,Y 69.08,Z 334.498,A -85,B 0,C 180,E1 -23620.911,E2 -23620.911} C_VEL
LIN {X 0,Y 68.037,Z 347.057,A -85,B 0,C 180,E1 -23617.78,E2 -23617.78} C_VEL
LIN {X 0,Y 66.87,Z 360.105,A -85,B 0,C 180,E1 -23613.143,E2 -23613.143} C_VEL
LIN {X 0,Y 65.881,Z 372.862,A -85,B 0,C 180,E1 -23606.951,E2 -23606.951} C_VEL
LIN {X 0,Y 65.514,Z 383.264,A -85,B 0,C 180,E1 -23600.401,E2 -23600.401} C_VEL
LIN {X 0,Y 65.872,Z 393.444,A -85,B 0,C 180,E1 -23592.318,E2 -23592.318} C_VEL
LIN {X 0,Y 67.82,Z 403.279,A -85,B 0,C 180,E1 -23582.967,E2 -23582.967} C_VEL
LIN {X 0,Y 71.602,Z 411.295,A -85,B 0,C 180,E1 -23574.364,E2 -23574.364} C_VEL
LIN {X 0,Y 76.964,Z 417.817,A -85,B 0,C 180,E1 -23566.801,E2 -23566.801} C_VEL
LIN {X 0,Y 83.714,Z 423.178,A -85,B 0,C 180,E1 -23560.376,E2 -23560.376} C_VEL
LIN {X 0,Y 91.594,Z 427.378,A -85,B 0,C 180,E1 -23555.033,E2 -23555.033} C_VEL
LIN {X 0,Y 102.609,Z 431.141,A -85,B 0,C 180,E1 -23549.697,E2 -23549.697} C_VEL
LIN {X 0,Y 103.671,Z 431.422,A -85,B 0,C 180,E1 -23549.275,E2 -23549.275} C_VEL
LIN {X 0,Y 102.028,Z 431.437,A -85,B 0,C 180,E1 -23547.937,E2 -23547.937} C_VEL
LIN {X 0,Y 94.901,Z 430.59,A -85,B 0,C 180,E1 -23544.554,E2 -23544.554} C_VEL
LIN {X 0,Y 85.095,Z 428.367,A -85,B 0,C 180,E1 -23538.018,E2 -23538.018} C_VEL
LIN {X 0,Y 77.175,Z 424.947,A -85,B 0,C 180,E1 -23529.607,E2 -23529.607} C_VEL
LIN {X 0,Y 71.76,Z 420.346,A -85,B 0,C 180,E1 -23519.324,E2 -23519.324} C_VEL
LIN {X 0,Y 69.595,Z 414.279,A -85,B 0,C 180,E1 -23507.639,E2 -23507.639} C_VEL
LIN {X 0,Y 70.293,Z 408.727,A -85,B 0,C 180,E1 -23498.629,E2 -23498.629} C_VEL
LIN {X 0,Y 69.942,Z 405.996,A -85,B 0,C 180,E1 -23495.771,E2 -23495.771} C_VEL
LIN {X 0,Y 68.691,Z 397.36,A -85,B 0,C 180,E1 -23488.538,E2 -23488.538} C_VEL
LIN {X 0,Y 68.358,Z 386.481,A -85,B 0,C 180,E1 -23481.133,E2 -23481.133} C_VEL
LIN {X 0,Y 68.866,Z 375.36,A -85,B 0,C 180,E1 -23475.223,E2 -23475.223} C_VEL
LIN {X 0,Y 69.165,Z 370.632,A -85,B 0,C 180,E1 -23473.148,E2 -23473.148} C_VEL
LIN {X 0,Y 68.836,Z 365.233,A -85,B 0,C 180,E1 -23471.165,E2 -23471.165} C_VEL
LIN {X 0,Y 67.581,Z 359.728,A -85,B 0,C 180,E1 -23469.557,E2 -23469.557} C_VEL
LIN {X 0,Y 64.193,Z 346.594,A -85,B 0,C 180,E1 -23466.538,E2 -23466.538} C_VEL
LIN {X 0,Y 63.877,Z 340.779,A -85,B 0,C 180,E1 -23465.378,E2 -23465.378} C_VEL
LIN {X 0,Y 65.474,Z 304.169,A -85,B 0,C 180,E1 -23458.808,E2 -23458.808} C_VEL
LIN {X 0,Y 64.468,Z 268.165,A -85,B 0,C 180,E1 -23452.421,E2 -23452.421} C_VEL
LIN {X 0,Y 64.4,Z 262.953,A -85,B 0,C 180,E1 -23451.485,E2 -23451.485} C_VEL
LIN {X 0,Y 60.871,Z 248.611,A -85,B 0,C 180,E1 -23448.147,E2 -23448.147} C_VEL
LIN {X 0,Y 59.414,Z 242.323,A -85,B 0,C 180,E1 -23440.59,E2 -23440.59} C_VEL
LIN {X 0,Y 58.182,Z 237.334,A -85,B 0,C 180,E1 -23433.669,E2 -23433.669} C_VEL
LIN {X 0,Y 58.15,Z 237.237,A -85,B 0,C 180,E1 -23428.914,E2 -23428.914} C_VEL
LIN {X 0,Y 58.522,Z 237.194,A -85,B 0,C 180,E1 -23416.128,E2 -23416.128} C_VEL
LIN {X 0,Y 58.813,Z 237.159,A -85,B 0,C 180,E1 -23406.866,E2 -23406.866} C_VEL
LIN {X 0,Y 59.379,Z 237.084,A -85,B 0,C 180,E1 -23400.003,E2 -23400.003} C_VEL
LIN {X 0,Y 58.793,Z 237.153,A -85,B 0,C 180,E1 -23393.138,E2 -23393.138} C_VEL
LIN {X 0,Y 58.511,Z 237.19,A -85,B 0,C 180,E1 -23383.909,E2 -23383.909} C_VEL
LIN {X 0,Y 58.151,Z 237.239,A -85,B 0,C 180,E1 -23371.094,E2 -23371.094} C_VEL
LIN {X 0,Y 58.065,Z 237.25,A -85,B 0,C 180,E1 -23362.762,E2 -23362.762} C_VEL
LIN {X 0,Y 58.087,Z 237.244,A -85,B 0,C 180,E1 -23353.457,E2 -23353.457} C_VEL
LIN {X 0,Y 58.069,Z 237.252,A -85,B 0,C 180,E1 -23347.232,E2 -23347.232} C_VEL
LIN {X 0,Y 58.153,Z 237.242,A -85,B 0,C 180,E1 -23338.903,E2 -23338.903} C_VEL
LIN {X 0,Y 58.533,Z 237.185,A -85,B 0,C 180,E1 -23326.16,E2 -23326.16} C_VEL
LIN {X 0,Y 58.816,Z 237.151,A -85,B 0,C 180,E1 -23316.858,E2 -23316.858} C_VEL
LIN {X 0,Y 59.391,Z 237.078,A -85,B 0,C 180,E1 -23309.995,E2 -23309.995} C_VEL
LIN {X 0,Y 58.822,Z 237.153,A -85,B 0,C 180,E1 -23303.133,E2 -23303.133} C_VEL
LIN {X 0,Y 58.532,Z 237.187,A -85,B 0,C 180,E1 -23293.845,E2 -23293.845} C_VEL
LIN {X 0,Y 58.34,Z 237.277,A -85,B 0,C 180,E1 -23286.946,E2 -23286.946} C_VEL
LIN {X 0,Y 58.885,Z 239.417,A -85,B 0,C 180,E1 -23283.407,E2 -23283.407} C_VEL
LIN {X 0,Y 59.873,Z 243.508,A -85,B 0,C 180,E1 -23278.357,E2 -23278.357} C_VEL
LIN {X 0,Y 65.268,Z 265.646,A -85,B 0,C 180,E1 -23273.199,E2 -23273.199} C_VEL
LIN {X 0,Y 65.782,Z 273.424,A -85,B 0,C 180,E1 -23271.744,E2 -23271.744} C_VEL
LIN {X 0,Y 61.992,Z 334.488,A -85,B 0,C 180,E1 -23260.41,E2 -23260.41} C_VEL
LIN {X 0,Y 60.968,Z 346.859,A -85,B 0,C 180,E1 -23257.029,E2 -23257.029} C_VEL
LIN {X 0,Y 59.921,Z 359.052,A -85,B 0,C 180,E1 -23252.308,E2 -23252.308} C_VEL
LIN {X 0,Y 59.053,Z 371.676,A -85,B 0,C 180,E1 -23245.554,E2 -23245.554} C_VEL
LIN {X 0,Y 58.881,Z 382.659,A -85,B 0,C 180,E1 -23237.943,E2 -23237.943} C_VEL
LIN {X 0,Y 59.623,Z 393.561,A -85,B 0,C 180,E1 -23228.47,E2 -23228.47} C_VEL
LIN {X 0,Y 61.723,Z 401.899,A -85,B 0,C 180,E1 -23219.997,E2 -23219.997} C_VEL
LIN {X 0,Y 66.034,Z 410.187,A -85,B 0,C 180,E1 -23210.811,E2 -23210.811} C_VEL
LIN {X 0,Y 71.93,Z 417.049,A -85,B 0,C 180,E1 -23202.953,E2 -23202.953} C_VEL
LIN {X 0,Y 79.251,Z 422.633,A -85,B 0,C 180,E1 -23196.478,E2 -23196.478} C_VEL
LIN {X 0,Y 88.627,Z 427.561,A -85,B 0,C 180,E1 -23190.73,E2 -23190.73} C_VEL
LIN {X 0,Y 91.735,Z 428.825,A -85,B 0,C 180,E1 -23189.223,E2 -23189.223} C_VEL
LIN {X 0,Y 91.076,Z 428.887,A -85,B 0,C 180,E1 -23188.089,E2 -23188.089} C_VEL
LIN {X 0,Y 80.711,Z 426.255,A -85,B 0,C 180,E1 -23181.604,E2 -23181.604} C_VEL
LIN {X 0,Y 72.15,Z 422.492,A -85,B 0,C 180,E1 -23172.994,E2 -23172.994} C_VEL
LIN {X 0,Y 66.017,Z 417.244,A -85,B 0,C 180,E1 -23161.602,E2 -23161.602} C_VEL
LIN {X 0,Y 63.598,Z 411.064,A -85,B 0,C 180,E1 -23149.366,E2 -23149.366} C_VEL
LIN {X 0,Y 64.115,Z 405.014,A -85,B 0,C 180,E1 -23139.393,E2 -23139.393} C_VEL
LIN {X 0,Y 62.452,Z 396.602,A -85,B 0,C 180,E1 -23131.617,E2 -23131.617} C_VEL
LIN {X 0,Y 61.702,Z 386.984,A -85,B 0,C 180,E1 -23124.285,E2 -23124.285} C_VEL
LIN {X 0,Y 61.883,Z 377.798,A -85,B 0,C 180,E1 -23118.541,E2 -23118.541} C_VEL
LIN {X 0,Y 62.52,Z 366.017,A -85,B 0,C 180,E1 -23112.842,E2 -23112.842} C_VEL
LIN {X 0,Y 63.403,Z 353.703,A -85,B 0,C 180,E1 -23108.463,E2 -23108.463} C_VEL
LIN {X 0,Y 63.877,Z 340.779,A -85,B 0,C 180,E1 -23105.378,E2 -23105.378} C_VEL
LIN {X 0,Y 63.57,Z 335.008,A -85,B 0,C 180,E1 -23104.327,E2 -23104.327} C_VEL
LIN {X 0,Y 58.654,Z 316.091,A -85,B 0,C 180,E1 -23101.043,E2 -23101.043} C_VEL
LIN {X 0,Y 58.208,Z 310.293,A -85,B 0,C 180,E1 -23099.918,E2 -23099.918} C_VEL
LIN {X 0,Y 58.281,Z 302.57,A -85,B 0,C 180,E1 -23098.396,E2 -23098.396} C_VEL
LIN {X 0,Y 57.468,Z 267.619,A -85,B 0,C 180,E1 -23091.451,E2 -23091.451} C_VEL
LIN {X 0,Y 57.33,Z 263.567,A -85,B 0,C 180,E1 -23090.629,E2 -23090.629} C_VEL
LIN {X 0,Y 53.545,Z 248.405,A -85,B 0,C 180,E1 -23086.627,E2 -23086.627} C_VEL
LIN {X 0,Y 52.022,Z 241.899,A -85,B 0,C 180,E1 -23077.673,E2 -23077.673} C_VEL
LIN {X 0,Y 51.13,Z 238.216,A -85,B 0,C 180,E1 -23071.608,E2 -23071.608} C_VEL
LIN {X 0,Y 51.389,Z 238.079,A -85,B 0,C 180,E1 -23056.822,E2 -23056.822} C_VEL
LIN {X 0,Y 51.688,Z 238.044,A -85,B 0,C 180,E1 -23047.818,E2 -23047.818} C_VEL
LIN {X 0,Y 52.262,Z 237.97,A -85,B 0,C 180,E1 -23040.004,E2 -23040.004} C_VEL
LIN {X 0,Y 51.67,Z 238.042,A -85,B 0,C 180,E1 -23032.186,E2 -23032.186} C_VEL
LIN {X 0,Y 51.381,Z 238.08,A -85,B 0,C 180,E1 -23023.211,E2 -23023.211} C_VEL
LIN {X 0,Y 51.021,Z 238.122,A -85,B 0,C 180,E1 -23015.595,E2 -23015.595} C_VEL
LIN {X 0,Y 51.044,Z 238.124,A -85,B 0,C 180,E1 -23005.691,E2 -23005.691} C_VEL
LIN {X 0,Y 51.05,Z 238.126,A -85,B 0,C 180,E1 -22996.506,E2 -22996.506} C_VEL
LIN {X 0,Y 51.051,Z 238.12,A -85,B 0,C 180,E1 -22993.489,E2 -22993.489} C_VEL
LIN {X 0,Y 51.069,Z 238.114,A -85,B 0,C 180,E1 -22983.392,E2 -22983.392} C_VEL
LIN {X 0,Y 51.025,Z 238.12,A -85,B 0,C 180,E1 -22974.4,E2 -22974.4} C_VEL
LIN {X 0,Y 51.478,Z 238.064,A -85,B 0,C 180,E1 -22965.84,E2 -22965.84} C_VEL
LIN {X 0,Y 51.692,Z 238.037,A -85,B 0,C 180,E1 -22957.808,E2 -22957.808} C_VEL
LIN {X 0,Y 52.276,Z 237.964,A -85,B 0,C 180,E1 -22949.995,E2 -22949.995} C_VEL
LIN {X 0,Y 51.698,Z 238.037,A -85,B 0,C 180,E1 -22942.181,E2 -22942.181} C_VEL
LIN {X 0,Y 51.433,Z 238.071,A -85,B 0,C 180,E1 -22933.025,E2 -22933.025} C_VEL
LIN {X 0,Y 51.306,Z 238.176,A -85,B 0,C 180,E1 -22928.88,E2 -22928.88} C_VEL
LIN {X 0,Y 51.643,Z 239.659,A -85,B 0,C 180,E1 -22925.899,E2 -22925.899} C_VEL
LIN {X 0,Y 52.64,Z 243.799,A -85,B 0,C 180,E1 -22919.95,E2 -22919.95} C_VEL
LIN {X 0,Y 56.67,Z 259.976,A -85,B 0,C 180,E1 -22915.505,E2 -22915.505} C_VEL
LIN {X 0,Y 58.396,Z 268.11,A -85,B 0,C 180,E1 -22913.608,E2 -22913.608} C_VEL
LIN {X 0,Y 58.71,Z 273.656,A -85,B 0,C 180,E1 -22912.467,E2 -22912.467} C_VEL
LIN {X 0,Y 54.948,Z 333.835,A -85,B 0,C 180,E1 -22899.871,E2 -22899.871} C_VEL
LIN {X 0,Y 53.92,Z 346.601,A -85,B 0,C 180,E1 -22895.963,E2 -22895.963} C_VEL
LIN {X 0,Y 52.859,Z 360.105,A -85,B 0,C 180,E1 -22889.902,E2 -22889.902} C_VEL
LIN {X 0,Y 52.276,Z 371.836,A -85,B 0,C 180,E1 -22882.719,E2 -22882.719} C_VEL
LIN {X 0,Y 52.348,Z 382.337,A -85,B 0,C 180,E1 -22874.576,E2 -22874.576} C_VEL
LIN {X 0,Y 53.36,Z 391.7,A -85,B 0,C 180,E1 -22865.665,E2 -22865.665} C_VEL
LIN {X 0,Y 56.452,Z 401.649,A -85,B 0,C 180,E1 -22854.895,E2 -22854.895} C_VEL
LIN {X 0,Y 61.779,Z 410.264,A -85,B 0,C 180,E1 -22845.166,E2 -22845.166} C_VEL
LIN {X 0,Y 69.816,Z 418.172,A -85,B 0,C 180,E1 -22836.253,E2 -22836.253} C_VEL
LIN {X 0,Y 78.082,Z 423.696,A -85,B 0,C 180,E1 -22830.325,E2 -22830.325} C_VEL
LIN {X 0,Y 81.067,Z 425.327,A -85,B 0,C 180,E1 -22828.654,E2 -22828.654} C_VEL
LIN {X 0,Y 71.839,Z 422.039,A -85,B 0,C 180,E1 -22821.508,E2 -22821.508} C_VEL
LIN {X 0,Y 63.748,Z 417.293,A -85,B 0,C 180,E1 -22811.418,E2 -22811.418} C_VEL
LIN {X 0,Y 58.802,Z 411.202,A -85,B 0,C 180,E1 -22798.565,E2 -22798.565} C_VEL
LIN {X 0,Y 57.769,Z 404.679,A -85,B 0,C 180,E1 -22785.891,E2 -22785.891} C_VEL
LIN {X 0,Y 58.045,Z 402.599,A -85,B 0,C 180,E1 -22782.417,E2 -22782.417} C_VEL
LIN {X 0,Y 56.82,Z 397.507,A -85,B 0,C 180,E1 -22777.11,E2 -22777.11} C_VEL
LIN {X 0,Y 55.475,Z 388.363,A -85,B 0,C 180,E1 -22769.098,E2 -22769.098} C_VEL
LIN {X 0,Y 55.206,Z 378.375,A -85,B 0,C 180,E1 -22761.771,E2 -22761.771} C_VEL
LIN {X 0,Y 55.552,Z 367.197,A -85,B 0,C 180,E1 -22755.349,E2 -22755.349} C_VEL
LIN {X 0,Y 56.352,Z 354.514,A -85,B 0,C 180,E1 -22749.948,E2 -22749.948} C_VEL
LIN {X 0,Y 56.778,Z 341.422,A -85,B 0,C 180,E1 -22746.285,E2 -22746.285} C_VEL
LIN {X 0,Y 58.208,Z 310.293,A -85,B 0,C 180,E1 -22739.918,E2 -22739.918} C_VEL
LIN {X 0,Y 57.996,Z 306.447,A -85,B 0,C 180,E1 -22739.154,E2 -22739.154} C_VEL
LIN {X 0,Y 56.654,Z 300.798,A -85,B 0,C 180,E1 -22737.991,E2 -22737.991} C_VEL
LIN {X 0,Y 51.327,Z 286.08,A -85,B 0,C 180,E1 -22734.658,E2 -22734.658} C_VEL
LIN {X 0,Y 50.424,Z 280.324,A -85,B 0,C 180,E1 -22733.298,E2 -22733.298} C_VEL
LIN {X 0,Y 50.367,Z 264.728,A -85,B 0,C 180,E1 -22729.726,E2 -22729.726} C_VEL
LIN {X 0,Y 46.121,Z 247.832,A -85,B 0,C 180,E1 -22724.428,E2 -22724.428} C_VEL
LIN {X 0,Y 44.885,Z 242.648,A -85,B 0,C 180,E1 -22715.962,E2 -22715.962} C_VEL
LIN {X 0,Y 44.062,Z 239.073,A -85,B 0,C 180,E1 -22708.919,E2 -22708.919} C_VEL
LIN {X 0,Y 44.228,Z 238.968,A -85,B 0,C 180,E1 -22697.579,E2 -22697.579} C_VEL
LIN {X 0,Y 44.538,Z 238.929,A -85,B 0,C 180,E1 -22689.083,E2 -22689.083} C_VEL
LIN {X 0,Y 45.136,Z 238.857,A -85,B 0,C 180,E1 -22680.004,E2 -22680.004} C_VEL
LIN {X 0,Y 44.524,Z 238.936,A -85,B 0,C 180,E1 -22670.922,E2 -22670.922} C_VEL
LIN {X 0,Y 44.148,Z 238.986,A -85,B 0,C 180,E1 -22661.439,E2 -22661.439} C_VEL
LIN {X 0,Y 43.849,Z 239.02,A -85,B 0,C 180,E1 -22651.265,E2 -22651.265} C_VEL
LIN {X 0,Y 43.861,Z 239.012,A -85,B 0,C 180,E1 -22640.144,E2 -22640.144} C_VEL
LIN {X 0,Y 43.884,Z 239.018,A -85,B 0,C 180,E1 -22626.807,E2 -22626.807} C_VEL
LIN {X 0,Y 43.852,Z 239.023,A -85,B 0,C 180,E1 -22618.73,E2 -22618.73} C_VEL
LIN {X 0,Y 44.254,Z 238.964,A -85,B 0,C 180,E1 -22607.675,E2 -22607.675} C_VEL
LIN {X 0,Y 44.546,Z 238.927,A -85,B 0,C 180,E1 -22599.071,E2 -22599.071} C_VEL
LIN {X 0,Y 45.151,Z 238.851,A -85,B 0,C 180,E1 -22589.994,E2 -22589.994} C_VEL
LIN {X 0,Y 44.552,Z 238.926,A -85,B 0,C 180,E1 -22580.917,E2 -22580.917} C_VEL
LIN {X 0,Y 44.342,Z 239.01,A -85,B 0,C 180,E1 -22571.512,E2 -22571.512} C_VEL
LIN {X 0,Y 44.44,Z 239.864,A -85,B 0,C 180,E1 -22569.149,E2 -22569.149} C_VEL
LIN {X 0,Y 45.414,Z 244.021,A -85,B 0,C 180,E1 -22562.018,E2 -22562.018} C_VEL
LIN {X 0,Y 48.494,Z 255.967,A -85,B 0,C 180,E1 -22557.996,E2 -22557.996} C_VEL
LIN {X 0,Y 51.469,Z 269.662,A -85,B 0,C 180,E1 -22554.219,E2 -22554.219} C_VEL
LIN {X 0,Y 51.57,Z 274.122,A -85,B 0,C 180,E1 -22553.185,E2 -22553.185} C_VEL
LIN {X 0,Y 47.94,Z 333.039,A -85,B 0,C 180,E1 -22539.004,E2 -22539.004} C_VEL
LIN {X 0,Y 46.986,Z 345.496,A -85,B 0,C 180,E1 -22534.763,E2 -22534.763} C_VEL
LIN {X 0,Y 46.222,Z 356.271,A -85,B 0,C 180,E1 -22529.609,E2 -22529.609} C_VEL
LIN {X 0,Y 45.662,Z 368.378,A -85,B 0,C 180,E1 -22521.802,E2 -22521.802} C_VEL
LIN {X 0,Y 45.887,Z 378.694,A -85,B 0,C 180,E1 -22513.277,E2 -22513.277} C_VEL
LIN {X 0,Y 47.331,Z 389.609,A -85,B 0,C 180,E1 -22502.123,E2 -22502.123} C_VEL
LIN {X 0,Y 50.345,Z 398.609,A -85,B 0,C 180,E1 -22491.972,E2 -22491.972} C_VEL
LIN {X 0,Y 55.969,Z 407.565,A -85,B 0,C 180,E1 -22481.7,E2 -22481.7} C_VEL
LIN {X 0,Y 64.512,Z 416.102,A -85,B 0,C 180,E1 -22472.416,E2 -22472.416} C_VEL
LIN {X 0,Y 70.495,Z 420.459,A -85,B 0,C 180,E1 -22468.094,E2 -22468.094} C_VEL
LIN {X 0,Y 61.079,Z 415.612,A -85,B 0,C 180,E1 -22458.417,E2 -22458.417} C_VEL
LIN {X 0,Y 54.777,Z 409.954,A -85,B 0,C 180,E1 -22446.393,E2 -22446.393} C_VEL
LIN {X 0,Y 52.037,Z 402.755,A -85,B 0,C 180,E1 -22431.389,E2 -22431.389} C_VEL
LIN {X 0,Y 52.121,Z 399.791,A -85,B 0,C 180,E1 -22425.651,E2 -22425.651} C_VEL
LIN {X 0,Y 51.261,Z 396.544,A -85,B 0,C 180,E1 -22421.877,E2 -22421.877} C_VEL
LIN {X 0,Y 49.413,Z 387.411,A -85,B 0,C 180,E1 -22413.064,E2 -22413.064} C_VEL
LIN {X 0,Y 48.741,Z 377.401,A -85,B 0,C 180,E1 -22404.835,E2 -22404.835} C_VEL
LIN {X 0,Y 48.818,Z 366.132,A -85,B 0,C 180,E1 -22397.535,E2 -22397.535} C_VEL
LIN {X 0,Y 49.468,Z 353.32,A -85,B 0,C 180,E1 -22391.364,E2 -22391.364} C_VEL
LIN {X 0,Y 49.811,Z 340.103,A -85,B 0,C 180,E1 -22387.176,E2 -22387.176} C_VEL
LIN {X 0,Y 51.287,Z 304.508,A -85,B 0,C 180,E1 -22378.798,E2 -22378.798} C_VEL
LIN {X 0,Y 50.424,Z 280.324,A -85,B 0,C 180,E1 -22373.298,E2 -22373.298} C_VEL
LIN {X 0,Y 49.518,Z 274.604,A -85,B 0,C 180,E1 -22371.884,E2 -22371.884} C_VEL
LIN {X 0,Y 47.567,Z 269.128,A -85,B 0,C 180,E1 -22370.314,E2 -22370.314} C_VEL
LIN {X 0,Y 40.948,Z 254.95,A -85,B 0,C 180,E1 -22365.139,E2 -22365.139} C_VEL
LIN {X 0,Y 39.733,Z 251.235,A -85,B 0,C 180,E1 -22363.676,E2 -22363.676} C_VEL
LIN {X 0,Y 38.724,Z 247.376,A -85,B 0,C 180,E1 -22361.622,E2 -22361.622} C_VEL
LIN {X 0,Y 37.505,Z 242.108,A -85,B 0,C 180,E1 -22351.025,E2 -22351.025} C_VEL
LIN {X 0,Y 36.898,Z 239.977,A -85,B 0,C 180,E1 -22345.382,E2 -22345.382} C_VEL
LIN {X 0,Y 37.069,Z 239.858,A -85,B 0,C 180,E1 -22338.592,E2 -22338.592} C_VEL
LIN {X 0,Y 37.332,Z 239.825,A -85,B 0,C 180,E1 -22330.856,E2 -22330.856} C_VEL
LIN {X 0,Y 37.994,Z 239.746,A -85,B 0,C 180,E1 -22320.005,E2 -22320.005} C_VEL
LIN {X 0,Y 37.321,Z 239.836,A -85,B 0,C 180,E1 -22309.151,E2 -22309.151} C_VEL
LIN {X 0,Y 37.051,Z 239.87,A -85,B 0,C 180,E1 -22301.494,E2 -22301.494} C_VEL
LIN {X 0,Y 36.749,Z 239.906,A -85,B 0,C 180,E1 -22284.996,E2 -22284.996} C_VEL
LIN {X 0,Y 36.772,Z 239.895,A -85,B 0,C 180,E1 -22279.85,E2 -22279.85} C_VEL
LIN {X 0,Y 36.773,Z 239.896,A -85,B 0,C 180,E1 -22270.148,E2 -22270.148} C_VEL
LIN {X 0,Y 36.75,Z 239.899,A -85,B 0,C 180,E1 -22265,E2 -22265} C_VEL
LIN {X 0,Y 37.077,Z 239.86,A -85,B 0,C 180,E1 -22248.62,E2 -22248.62} C_VEL
LIN {X 0,Y 37.344,Z 239.829,A -85,B 0,C 180,E1 -22240.84,E2 -22240.84} C_VEL
LIN {X 0,Y 38.01,Z 239.741,A -85,B 0,C 180,E1 -22229.993,E2 -22229.993} C_VEL
LIN {X 0,Y 37.273,Z 239.921,A -85,B 0,C 180,E1 -22214.614,E2 -22214.614} C_VEL
LIN {X 0,Y 37.763,Z 242.502,A -85,B 0,C 180,E1 -22208.14,E2 -22208.14} C_VEL
LIN {X 0,Y 38.238,Z 244.514,A -85,B 0,C 180,E1 -22204.479,E2 -22204.479} C_VEL
LIN {X 0,Y 41.349,Z 256.161,A -85,B 0,C 180,E1 -22199.724,E2 -22199.724} C_VEL
LIN {X 0,Y 44.483,Z 270.615,A -85,B 0,C 180,E1 -22195.047,E2 -22195.047} C_VEL
LIN {X 0,Y 44.457,Z 274.629,A -85,B 0,C 180,E1 -22193.984,E2 -22193.984} C_VEL
LIN {X 0,Y 40.937,Z 332.616,A -85,B 0,C 180,E1 -22177.699,E2 -22177.699} C_VEL
LIN {X 0,Y 40.051,Z 344.935,A -85,B 0,C 180,E1 -22172.874,E2 -22172.874} C_VEL
LIN {X 0,Y 39.392,Z 356.163,A -85,B 0,C 180,E1 -22166.533,E2 -22166.533} C_VEL
LIN {X 0,Y 39.228,Z 368.711,A -85,B 0,C 180,E1 -22156.921,E2 -22156.921} C_VEL
LIN {X 0,Y 39.896,Z 378.427,A -85,B 0,C 180,E1 -22147.587,E2 -22147.587} C_VEL
LIN {X 0,Y 42.004,Z 388.904,A -85,B 0,C 180,E1 -22135.787,E2 -22135.787} C_VEL
LIN {X 0,Y 46.19,Z 398.368,A -85,B 0,C 180,E1 -22124.535,E2 -22124.535} C_VEL
LIN {X 0,Y 52.911,Z 407.39,A -85,B 0,C 180,E1 -22114.419,E2 -22114.419} C_VEL
LIN {X 0,Y 60.073,Z 414.155,A -85,B 0,C 180,E1 -22107.585,E2 -22107.585} C_VEL
LIN {X 0,Y 59.412,Z 413.924,A -85,B 0,C 180,E1 -22105.906,E2 -22105.906} C_VEL
LIN {X 0,Y 51.142,Z 407.725,A -85,B 0,C 180,E1 -22093.409,E2 -22093.409} C_VEL
LIN {X 0,Y 47.057,Z 401.129,A -85,B 0,C 180,E1 -22079.045,E2 -22079.045} C_VEL
LIN {X 0,Y 46.387,Z 396.016,A -85,B 0,C 180,E1 -22068.567,E2 -22068.567} C_VEL
LIN {X 0,Y 43.861,Z 387.413,A -85,B 0,C 180,E1 -22059.227,E2 -22059.227} C_VEL
LIN {X 0,Y 42.443,Z 376.375,A -85,B 0,C 180,E1 -22048.792,E2 -22048.792} C_VEL
LIN {X 0,Y 42.206,Z 365.1,A -85,B 0,C 180,E1 -22040.421,E2 -22040.421} C_VEL
LIN {X 0,Y 42.593,Z 353.457,A -85,B 0,C 180,E1 -22033.84,E2 -22033.84} C_VEL
LIN {X 0,Y 42.836,Z 340.662,A -85,B 0,C 180,E1 -22028.975,E2 -22028.975} C_VEL
LIN {X 0,Y 44.222,Z 304.824,A -85,B 0,C 180,E1 -22019.07,E2 -22019.07} C_VEL
LIN {X 0,Y 43.359,Z 269.082,A -85,B 0,C 180,E1 -22009.592,E2 -22009.592} C_VEL
LIN {X 0,Y 43.314,Z 265.597,A -85,B 0,C 180,E1 -22008.649,E2 -22008.649} C_VEL
LIN {X 0,Y 39.733,Z 251.235,A -85,B 0,C 180,E1 -22003.676,E2 -22003.676} C_VEL
LIN {X 0,Y 38.417,Z 248.769,A -85,B 0,C 180,E1 -22001.987,E2 -22001.987} C_VEL
LIN {X 0,Y 35.674,Z 246.368,A -85,B 0,C 180,E1 -21998.172,E2 -21998.172} C_VEL
LIN {X 0,Y 30.653,Z 242.064,A -85,B 0,C 180,E1 -21985.275,E2 -21985.275} C_VEL
LIN {X 0,Y 30.015,Z 240.733,A -85,B 0,C 180,E1 -21978.765,E2 -21978.765} C_VEL
LIN {X 0,Y 30.018,Z 240.659,A -85,B 0,C 180,E1 -21977.35,E2 -21977.35} C_VEL
LIN {X 0,Y 30.811,Z 240.549,A -85,B 0,C 180,E1 -21960.006,E2 -21960.006} C_VEL
LIN {X 0,Y 30.1,Z 240.615,A -85,B 0,C 180,E1 -21946.504,E2 -21946.504} C_VEL
LIN {X 0,Y 29.86,Z 240.639,A -85,B 0,C 180,E1 -21940.268,E2 -21940.268} C_VEL
LIN {X 0,Y 29.506,Z 240.672,A -85,B 0,C 180,E1 -21931.558,E2 -21931.558} C_VEL
LIN {X 0,Y 29.592,Z 240.664,A -85,B 0,C 180,E1 -21914.572,E2 -21914.572} C_VEL
LIN {X 0,Y 29.549,Z 240.669,A -85,B 0,C 180,E1 -21898.393,E2 -21898.393} C_VEL
LIN {X 0,Y 29.888,Z 240.637,A -85,B 0,C 180,E1 -21889.87,E2 -21889.87} C_VEL
LIN {X 0,Y 30.123,Z 240.615,A -85,B 0,C 180,E1 -21883.482,E2 -21883.482} C_VEL
LIN {X 0,Y 30.829,Z 240.546,A -85,B 0,C 180,E1 -21869.991,E2 -21869.991} C_VEL
LIN {X 0,Y 30.305,Z 240.828,A -85,B 0,C 180,E1 -21858.707,E2 -21858.707} C_VEL
LIN {X 0,Y 30.989,Z 244.554,A -85,B 0,C 180,E1 -21848.449,E2 -21848.449} C_VEL
LIN {X 0,Y 33.885,Z 254.864,A -85,B 0,C 180,E1 -21842.781,E2 -21842.781} C_VEL
LIN {X 0,Y 37.556,Z 272.376,A -85,B 0,C 180,E1 -21835.839,E2 -21835.839} C_VEL
LIN {X 0,Y 33.994,Z 332.08,A -85,B 0,C 180,E1 -21815.626,E2 -21815.626} C_VEL
LIN {X 0,Y 33.257,Z 344.212,A -85,B 0,C 180,E1 -21809.925,E2 -21809.925} C_VEL
LIN {X 0,Y 32.776,Z 356.937,A -85,B 0,C 180,E1 -21801.207,E2 -21801.207} C_VEL
LIN {X 0,Y 33.149,Z 368.468,A -85,B 0,C 180,E1 -21790.685,E2 -21790.685} C_VEL
LIN {X 0,Y 34.388,Z 378.093,A -85,B 0,C 180,E1 -21779.994,E2 -21779.994} C_VEL
LIN {X 0,Y 37.387,Z 388.006,A -85,B 0,C 180,E1 -21767.786,E2 -21767.786} C_VEL
LIN {X 0,Y 42.956,Z 397.987,A -85,B 0,C 180,E1 -21755.852,E2 -21755.852} C_VEL
LIN {X 0,Y 50.816,Z 407.16,A -85,B 0,C 180,E1 -21746.408,E2 -21746.408} C_VEL
LIN {X 0,Y 51.126,Z 407.519,A -85,B 0,C 180,E1 -21745.576,E2 -21745.576} C_VEL
LIN {X 0,Y 43.038,Z 399.228,A -85,B 0,C 180,E1 -21727.765,E2 -21727.765} C_VEL
LIN {X 0,Y 41.309,Z 393.947,A -85,B 0,C 180,E1 -21715.646,E2 -21715.646} C_VEL
LIN {X 0,Y 40.948,Z 392.427,A -85,B 0,C 180,E1 -21712.955,E2 -21712.955} C_VEL
LIN {X 0,Y 38.068,Z 383.928,A -85,B 0,C 180,E1 -21703.35,E2 -21703.35} C_VEL
LIN {X 0,Y 36.466,Z 374.495,A -85,B 0,C 180,E1 -21693.603,E2 -21693.603} C_VEL
LIN {X 0,Y 35.758,Z 362.59,A -85,B 0,C 180,E1 -21683.477,E2 -21683.477} C_VEL
LIN {X 0,Y 35.849,Z 350.567,A -85,B 0,C 180,E1 -21675.823,E2 -21675.823} C_VEL
LIN {X 0,Y 35.972,Z 337.984,A -85,B 0,C 180,E1 -21670.387,E2 -21670.387} C_VEL
LIN {X 0,Y 37.079,Z 304.247,A -85,B 0,C 180,E1 -21659.189,E2 -21659.189} C_VEL
LIN {X 0,Y 36.213,Z 266.276,A -85,B 0,C 180,E1 -21647.174,E2 -21647.174} C_VEL
LIN {X 0,Y 32.173,Z 249.85,A -85,B 0,C 180,E1 -21639.925,E2 -21639.925} C_VEL
LIN {X 0,Y 31.384,Z 247.111,A -85,B 0,C 180,E1 -21638.02,E2 -21638.02} C_VEL
LIN {X 0,Y 30.396,Z 243.009,A -85,B 0,C 180,E1 -21627.551,E2 -21627.551} C_VEL
LIN {X 0,Y 29.943,Z 240.72,A -85,B 0,C 180,E1 -21620.169,E2 -21620.169} C_VEL
LIN {X 0,Y 30.018,Z 240.659,A -85,B 0,C 180,E1 -21617.35,E2 -21617.35} C_VEL
LIN {X 0,Y 29.582,Z 240.664,A -85,B 0,C 180,E1 -21611.258,E2 -21611.258} C_VEL
LIN {X 0,Y 27.818,Z 240.834,A -85,B 0,C 180,E1 -21602.799,E2 -21602.799} C_VEL
LIN {X 0,Y 25.092,Z 241.014,A -85,B 0,C 180,E1 -21592.284,E2 -21592.284} C_VEL
LIN {X 0,Y 22.213,Z 241.076,A -85,B 0,C 180,E1 -21572.243,E2 -21572.243} C_VEL
LIN {X 0,Y 22.22,Z 241.084,A -85,B 0,C 180,E1 -21560.771,E2 -21560.771} C_VEL
LIN {X 0,Y 22.233,Z 241.083,A -85,B 0,C 180,E1 -21549.197,E2 -21549.197} C_VEL
LIN {X 0,Y 22.839,Z 241.064,A -85,B 0,C 180,E1 -21527.908,E2 -21527.908} C_VEL
LIN {X 0,Y 23.571,Z 241.133,A -85,B 0,C 180,E1 -21508.92,E2 -21508.92} C_VEL
LIN {X 0,Y 23.871,Z 244.719,A -85,B 0,C 180,E1 -21494.513,E2 -21494.513} C_VEL
LIN {X 0,Y 25.431,Z 249.962,A -85,B 0,C 180,E1 -21489.618,E2 -21489.618} C_VEL
LIN {X 0,Y 28.223,Z 261.704,A -85,B 0,C 180,E1 -21482.595,E2 -21482.595} C_VEL
LIN {X 0,Y 30.502,Z 272.826,A -85,B 0,C 180,E1 -21477.252,E2 -21477.252} C_VEL
LIN {X 0,Y 27.137,Z 331.698,A -85,B 0,C 180,E1 -21452.246,E2 -21452.246} C_VEL
LIN {X 0,Y 26.561,Z 344.145,A -85,B 0,C 180,E1 -21444.934,E2 -21444.934} C_VEL
LIN {X 0,Y 26.543,Z 356.603,A -85,B 0,C 180,E1 -21434.365,E2 -21434.365} C_VEL
LIN {X 0,Y 27.642,Z 368.1,A -85,B 0,C 180,E1 -21421.814,E2 -21421.814} C_VEL
LIN {X 0,Y 30.092,Z 378.38,A -85,B 0,C 180,E1 -21408.737,E2 -21408.737} C_VEL
LIN {X 0,Y 34.559,Z 388.47,A -85,B 0,C 180,E1 -21395.995,E2 -21395.995} C_VEL
LIN {X 0,Y 40.864,Z 397.578,A -85,B 0,C 180,E1 -21386.011,E2 -21386.011} C_VEL
LIN {X 0,Y 42.287,Z 399.199,A -85,B 0,C 180,E1 -21384.424,E2 -21384.424} C_VEL
LIN {X 0,Y 41.072,Z 398.083,A -85,B 0,C 180,E1 -21379.895,E2 -21379.895} C_VEL
LIN {X 0,Y 36.601,Z 390.636,A -85,B 0,C 180,E1 -21362.162,E2 -21362.162} C_VEL
LIN {X 0,Y 36.192,Z 389.373,A -85,B 0,C 180,E1 -21359.604,E2 -21359.604} C_VEL
LIN {X 0,Y 32.535,Z 380.202,A -85,B 0,C 180,E1 -21348.915,E2 -21348.915} C_VEL
LIN {X 0,Y 30.51,Z 370.735,A -85,B 0,C 180,E1 -21338.287,E2 -21338.287} C_VEL
LIN {X 0,Y 29.466,Z 359.566,A -85,B 0,C 180,E1 -21327.704,E2 -21327.704} C_VEL
LIN {X 0,Y 29.27,Z 348.819,A -85,B 0,C 180,E1 -21319.692,E2 -21319.692} C_VEL
LIN {X 0,Y 29.145,Z 335.65,A -85,B 0,C 180,E1 -21313.028,E2 -21313.028} C_VEL
LIN {X 0,Y 30.011,Z 304.403,A -85,B 0,C 180,E1 -21300.047,E2 -21300.047} C_VEL
LIN {X 0,Y 29.266,Z 267.459,A -85,B 0,C 180,E1 -21285.482,E2 -21285.482} C_VEL
LIN {X 0,Y 25.461,Z 251.597,A -85,B 0,C 180,E1 -21276.535,E2 -21276.535} C_VEL
LIN {X 0,Y 24.069,Z 246.966,A -85,B 0,C 180,E1 -21272.555,E2 -21272.555} C_VEL
LIN {X 0,Y 23.211,Z 242.683,A -85,B 0,C 180,E1 -21257.634,E2 -21257.634} C_VEL
LIN {X 0,Y 23.068,Z 241.158,A -85,B 0,C 180,E1 -21249.876,E2 -21249.876} C_VEL
LIN {X 0,Y 23.581,Z 241.048,A -85,B 0,C 180,E1 -21240.008,E2 -21240.008} C_VEL
LIN {X 0,Y 22.811,Z 241.065,A -85,B 0,C 180,E1 -21222.064,E2 -21222.064} C_VEL
LIN {X 0,Y 22.213,Z 241.076,A -85,B 0,C 180,E1 -21212.243,E2 -21212.243} C_VEL
LIN {X 0,Y 21.34,Z 241.113,A -85,B 0,C 180,E1 -21201.803,E2 -21201.803} C_VEL
LIN {X 0,Y 19.957,Z 241.154,A -85,B 0,C 180,E1 -21190.99,E2 -21190.99} C_VEL
LIN {X 0,Y 18.106,Z 241.602,A -85,B 0,C 180,E1 -21175.017,E2 -21175.017} C_VEL
LIN {X 0,Y 17.034,Z 243.035,A -85,B 0,C 180,E1 -21157.368,E2 -21157.368} C_VEL
LIN {X 0,Y 16.939,Z 244.321,A -85,B 0,C 180,E1 -21148.868,E2 -21148.868} C_VEL
LIN {X 0,Y 17.109,Z 245.726,A -85,B 0,C 180,E1 -21143.349,E2 -21143.349} C_VEL
LIN {X 0,Y 19.738,Z 254.877,A -85,B 0,C 180,E1 -21132.502,E2 -21132.502} C_VEL
LIN {X 0,Y 23.434,Z 272.906,A -85,B 0,C 180,E1 -21119.583,E2 -21119.583} C_VEL
LIN {X 0,Y 20.453,Z 330.991,A -85,B 0,C 180,E1 -21086.797,E2 -21086.797} C_VEL
LIN {X 0,Y 20.269,Z 344.609,A -85,B 0,C 180,E1 -21075.966,E2 -21075.966} C_VEL
LIN {X 0,Y 21.107,Z 356.947,A -85,B 0,C 180,E1 -21062.359,E2 -21062.359} C_VEL
LIN {X 0,Y 23.222,Z 367.665,A -85,B 0,C 180,E1 -21048.772,E2 -21048.772} C_VEL
LIN {X 0,Y 26.509,Z 376.959,A -85,B 0,C 180,E1 -21036.559,E2 -21036.559} C_VEL
LIN {X 0,Y 31.349,Z 385.881,A -85,B 0,C 180,E1 -21025.905,E2 -21025.905} C_VEL
LIN {X 0,Y 35.071,Z 391.006,A -85,B 0,C 180,E1 -21020.679,E2 -21020.679} C_VEL
LIN {X 0,Y 32.629,Z 387.084,A -85,B 0,C 180,E1 -21010.264,E2 -21010.264} C_VEL
LIN {X 0,Y 31.847,Z 385.516,A -85,B 0,C 180,E1 -21007.374,E2 -21007.374} C_VEL
LIN {X 0,Y 27.116,Z 374.906,A -85,B 0,C 180,E1 -20994.92,E2 -20994.92} C_VEL
LIN {X 0,Y 24.499,Z 364.338,A -85,B 0,C 180,E1 -20982.436,E2 -20982.436} C_VEL
LIN {X 0,Y 23.17,Z 352.191,A -85,B 0,C 180,E1 -20970.012,E2 -20970.012} C_VEL
LIN {X 0,Y 22.617,Z 339.929,A -85,B 0,C 180,E1 -20960.963,E2 -20960.963} C_VEL
LIN {X 0,Y 22.957,Z 304.752,A -85,B 0,C 180,E1 -20941.624,E2 -20941.624} C_VEL
LIN {X 0,Y 22.214,Z 268.03,A -85,B 0,C 180,E1 -20922.561,E2 -20922.561} C_VEL
LIN {X 0,Y 18.891,Z 253.265,A -85,B 0,C 180,E1 -20910.699,E2 -20910.699} C_VEL
LIN {X 0,Y 16.84,Z 246.896,A -85,B 0,C 180,E1 -20902.235,E2 -20902.235} C_VEL
LIN {X 0,Y 16.596,Z 244.689,A -85,B 0,C 180,E1 -20892.236,E2 -20892.236} C_VEL
LIN {X 0,Y 16.469,Z 242.75,A -85,B 0,C 180,E1 -20880.012,E2 -20880.012} C_VEL
LIN {X 0,Y 15.676,Z 241.45,A -85,B 0,C 180,E1 -20863.362,E2 -20863.362} C_VEL
LIN {X 0,Y 15.025,Z 241.256,A -85,B 0,C 180,E1 -20837.141,E2 -20837.141} C_VEL
LIN {X 0,Y 15.038,Z 241.433,A -85,B 0,C 180,E1 -20823.686,E2 -20823.686} C_VEL
LIN {X 0,Y 15.925,Z 242.726,A -85,B 0,C 180,E1 -20802.729,E2 -20802.729} C_VEL
LIN {X 0,Y 16.939,Z 244.321,A -85,B 0,C 180,E1 -20788.868,E2 -20788.868} C_VEL
LIN {X 0,Y 17.877,Z 246.263,A -85,B 0,C 180,E1 -20781.577,E2 -20781.577} C_VEL
LIN {X 0,Y 20.542,Z 250.22,A -85,B 0,C 180,E1 -20774.429,E2 -20774.429} C_VEL
LIN {X 0,Y 21.996,Z 253.909,A -85,B 0,C 180,E1 -20770.619,E2 -20770.619} C_VEL
LIN {X 0,Y 22.379,Z 258.258,A -85,B 0,C 180,E1 -20767.926,E2 -20767.926} C_VEL
LIN {X 0,Y 21.405,Z 262.403,A -85,B 0,C 180,E1 -20766.927,E2 -20766.927} C_VEL
LIN {X 0,Y 17.015,Z 271.819,A -85,B 0,C 180,E1 -20764.059,E2 -20764.059} C_VEL
LIN {X 0,Y 16.269,Z 275.133,A -85,B 0,C 180,E1 -20762.098,E2 -20762.098} C_VEL
LIN {X 0,Y 14.263,Z 330.651,A -85,B 0,C 180,E1 -20715.147,E2 -20715.147} C_VEL
LIN {X 0,Y 14.878,Z 343.851,A -85,B 0,C 180,E1 -20700.833,E2 -20700.833} C_VEL
LIN {X 0,Y 16.633,Z 354.945,A -85,B 0,C 180,E1 -20686.596,E2 -20686.596} C_VEL
LIN {X 0,Y 20.33,Z 366.744,A -85,B 0,C 180,E1 -20671.608,E2 -20671.608} C_VEL
LIN {X 0,Y 25.439,Z 376.954,A -85,B 0,C 180,E1 -20659.884,E2 -20659.884} C_VEL
LIN {X 0,Y 26.417,Z 378.526,A -85,B 0,C 180,E1 -20658.3,E2 -20658.3} C_VEL
LIN {X 0,Y 25.778,Z 377.07,A -85,B 0,C 180,E1 -20652.983,E2 -20652.983} C_VEL
LIN {X 0,Y 21.611,Z 367.412,A -85,B 0,C 180,E1 -20641.916,E2 -20641.916} C_VEL
LIN {X 0,Y 18.702,Z 356.664,A -85,B 0,C 180,E1 -20629.212,E2 -20629.212} C_VEL
LIN {X 0,Y 17.139,Z 345.799,A -85,B 0,C 180,E1 -20617.379,E2 -20617.379} C_VEL
LIN {X 0,Y 15.883,Z 327.109,A -85,B 0,C 180,E1 -20602.399,E2 -20602.399} C_VEL
LIN {X 0,Y 15.9,Z 304.301,A -85,B 0,C 180,E1 -20584.304,E2 -20584.304} C_VEL
LIN {X 0,Y 15.41,Z 269.296,A -85,B 0,C 180,E1 -20557.94,E2 -20557.94} C_VEL
LIN {X 0,Y 12.597,Z 254.795,A -85,B 0,C 180,E1 -20539.362,E2 -20539.362} C_VEL
LIN {X 0,Y 11.001,Z 248.774,A -85,B 0,C 180,E1 -20524.598,E2 -20524.598} C_VEL
LIN {X 0,Y 10.214,Z 246.339,A -85,B 0,C 180,E1 -20513.033,E2 -20513.033} C_VEL
LIN {X 0,Y 9.726,Z 245.702,A -85,B 0,C 180,E1 -20500.106,E2 -20500.106} C_VEL
LIN {X 0,Y 9.437,Z 245.639,A -85,B 0,C 180,E1 -20469.153,E2 -20469.153} C_VEL
LIN {X 0,Y 10.899,Z 247.822,A -85,B 0,C 180,E1 -20442.98,E2 -20442.98} C_VEL
LIN {X 0,Y 11.765,Z 249.27,A -85,B 0,C 180,E1 -20435.959,E2 -20435.959} C_VEL
LIN {X 0,Y 13.656,Z 258.073,A -85,B 0,C 180,E1 -20419.789,E2 -20419.789} C_VEL
LIN {X 0,Y 16.414,Z 273.603,A -85,B 0,C 180,E1 -20403.112,E2 -20403.112} C_VEL
LIN {X 0,Y 16.269,Z 275.133,A -85,B 0,C 180,E1 -20402.098,E2 -20402.098} C_VEL
LIN {X 0,Y 15.135,Z 280.83,A -85,B 0,C 180,E1 -20398.457,E2 -20398.457} C_VEL
LIN {X 0,Y 11.492,Z 289.897,A -85,B 0,C 180,E1 -20391.433,E2 -20391.433} C_VEL
LIN {X 0,Y 8.011,Z 298.946,A -85,B 0,C 180,E1 -20377.98,E2 -20377.98} C_VEL
LIN {X 0,Y 7.225,Z 304.626,A -85,B 0,C 180,E1 -20366.588,E2 -20366.588} C_VEL
LIN {X 0,Y 9.416,Z 330.148,A -85,B 0,C 180,E1 -20329.311,E2 -20329.311} C_VEL
LIN {X 0,Y 11.664,Z 343.853,A -85,B 0,C 180,E1 -20312.47,E2 -20312.47} C_VEL
LIN {X 0,Y 15.128,Z 355.308,A -85,B 0,C 180,E1 -20300.282,E2 -20300.282} C_VEL
LIN {X 0,Y 16.518,Z 358.706,A -85,B 0,C 180,E1 -20296.727,E2 -20296.727} C_VEL
LIN {X 0,Y 16.618,Z 358.64,A -85,B 0,C 180,E1 -20293.375,E2 -20293.375} C_VEL
LIN {X 0,Y 13.271,Z 346.841,A -85,B 0,C 180,E1 -20280.89,E2 -20280.89} C_VEL
LIN {X 0,Y 11.019,Z 333.611,A -85,B 0,C 180,E1 -20268.624,E2 -20268.624} C_VEL
LIN {X 0,Y 9.064,Z 304.671,A -85,B 0,C 180,E1 -20233.209,E2 -20233.209} C_VEL
LIN {X 0,Y 8.664,Z 269.948,A -85,B 0,C 180,E1 -20185.97,E2 -20185.97} C_VEL
LIN {X 0,Y 7.57,Z 257.229,A -85,B 0,C 180,E1 -20153.114,E2 -20153.114} C_VEL
LIN {X 0,Y 7.637,Z 252.557,A -85,B 0,C 180,E1 -20133.177,E2 -20133.177} C_VEL
LIN {X 0,Y 7.598,Z 252.606,A -85,B 0,C 180,E1 -20114.266,E2 -20114.266} C_VEL
LIN {X 0,Y 7.825,Z 253.692,A -85,B 0,C 180,E1 -20100.892,E2 -20100.892} C_VEL
LIN {X 0,Y 8.126,Z 262.579,A -85,B 0,C 180,E1 -20074.465,E2 -20074.465} C_VEL
LIN {X 0,Y 9.418,Z 274.947,A -85,B 0,C 180,E1 -20050.3,E2 -20050.3} C_VEL
LIN {X 0,Y 7.225,Z 304.626,A -85,B 0,C 180,E1 -20006.588,E2 -20006.588} C_VEL
LIN {X 0,Y 6.297,Z 304.25,A -85,B 0,C 180,E1 -20003.426,E2 -20003.426} C_VEL
LIN {X 0,Y 5.39,Z 303.022,A -85,B 0,C 180,E1 -20001.337,E2 -20001.337} C_VEL
LIN {X 0,Y 2.53,Z 295.928,A -85,B 0,C 180,E1 -20001.956,E2 -20001.956} C_VEL
LIN {X 0,Y 0.796,Z 286.063,A -85,B 0,C 180,E1 -20103.565,E2 -20103.565} C_VEL
LIN {X 0,Y 1.961,Z 280.378,A -85,B 0,C 180,E1 -20137.321,E2 -20137.321} C_VEL
LIN {X 0,Y 3.153,Z 274.657,A -85,B 0,C 180,E1 -20137.733,E2 -20137.733} C_VEL
LIN {X 0,Y 3.865,Z 270.907,A -85,B 0,C 180,E1 -20132.65,E2 -20132.65} C_VEL
LIN {X 0,Y 4.315,Z 268.446,A -85,B 0,C 180,E1 -20122.46,E2 -20122.46} C_VEL
LIN {X 0,Y 4.184,Z 269.248,A -85,B 0,C 180,E1 -20116.073,E2 -20116.073} C_VEL
LIN {X 0,Y 3.518,Z 274.872,A -85,B 0,C 180,E1 -20091.165,E2 -20091.165} C_VEL
LIN {X 0,Y 3.984,Z 308.535,A -85,B 0,C 180,E1 -19929.277,E2 -19929.277} C_VEL
LIN {X 0,Y 4.094,Z 308.776,A -85,B 0,C 180,E1 -19926.304,E2 -19926.304} C_VEL
LIN {X 0,Y 2.697,Z 301.23,A -85,B 0,C 180,E1 -19914.415,E2 -19914.415} C_VEL
LIN {X 0,Y 3.153,Z 274.657,A -85,B 0,C 180,E1 -19777.733,E2 -19777.733} C_VEL
LIN {X 0,Y 7.069,Z 275.054,A -85,B 0,C 180,E1 -19770.599,E2 -19770.599} C_VEL
LIN {X 0,Y 7.069,Z 600,A -85,B 0,C 180,E1 -19770.599,E2 -19770.599} C_VEL
LIN {X 0,Y 7.069,Z 600,A -85,B 0,C 180,E1 -19770.599,E2 -19770.599}

QRS_NEXT_CUT()

QRS_NEXT()
QRS_HOME()

END
